// TwinCAT 3 PLC project PLC
// ProgramVersion: 3.1.4023.0
// libraries:
//   Tc2_Standard, * (Beckhoff Automation GmbH)
//   Tc2_System, * (Beckhoff Automation GmbH)
//   Tc3_Module, * (Beckhoff Automation GmbH)
// project tree:
//   / PlcTask.TcTTO
//   POUs/ MAIN.TcPOU
//   DUTs/IO/PdoEntries/ Status_57491DF1.TcDUT, Status_D4FDECD4.TcDUT, Control_0B2F8B70.TcDUT, Status_A3AA621F.TcDUT, Status_B0753356.TcDUT, Status_F2CE6D91.TcDUT, Status_7BCDA921.TcDUT, Ctrl_B9DDD3FF.TcDUT, STATUS_B0753356.TcDUT, Status_8F1D55D8.TcDUT, Status_ACC8459F.TcDUT, Status_3A9E406C.TcDUT, Control_D500AB79.TcDUT, Status_D8D782C3.TcDUT, Control_6EF2C5D0.TcDUT, Status_E2E79E85.TcDUT, Status_E3E7FD12.TcDUT, Status_8CBE219F.TcDUT, Status_B6795845.TcDUT, Control_5FD4673D.TcDUT, Status_1E008DB9.TcDUT, Status_3035BE2E.TcDUT, Control_F189B737.TcDUT, Control_C948E0F2.TcDUT, Status_725F98F2.TcDUT, Device_Diag_1464ECF9.TcDUT, Control_F58A89C5.TcDUT, Status_6CCA259F.TcDUT, Status_72C27E80.TcDUT, Control_254441A5.TcDUT, Status_15ACD201.TcDUT, Device_Status_033C68E9.TcDUT
//   DUTs/IO/PDOs/ InfoData_6F19DB2B.TcDUT, Channel_830843C1.TcDUT, WcState_9091E0EB.TcDUT, ID_Inputs_07C9D28F.TcDUT, InfoData_32EB74EA.TcDUT, Latch_8E413295.TcDUT, WcState_B516A264.TcDUT, InfoData_A7436BC6.TcDUT, CNT_Input_Channel_FF10BD3C.TcDUT, DIG_Inputs_CAFF6004.TcDUT, DIG_Inputs_Device_1F4E72EB.TcDUT, CNT_Output_Channel_550BB6DF.TcDUT, DI_X01_Pin_830843C1.TcDUT, DI_X02_Pin_830843C1.TcDUT, DI_X03_Pin_830843C1.TcDUT, DI_X04_Pin_830843C1.TcDUT, DI_X05_Pin_830843C1.TcDUT, DI_X06_Pin_830843C1.TcDUT, DI_X07_Pin_830843C1.TcDUT, DI_X08_Pin_830843C1.TcDUT, DI_X_830843C1.TcDUT, DIG_Inputs_Channel_ACAA0425.TcDUT, DO_Inputs_Channel_CC455148.TcDUT, DIG_Inputs_Channel_CC455148.TcDUT, DIG_Inputs_Channel_38F9DD27.TcDUT, DIG_Inputs_Device_B3EA4204.TcDUT, AI_Inputs_Channel_C3DE7A0A.TcDUT, DO_X05_Pin_42CA91F7.TcDUT, DO_X06_Pin_42CA91F7.TcDUT, DO_X07_Pin_42CA91F7.TcDUT, DO_X08_Pin_42CA91F7.TcDUT, DO_X_42CA91F7.TcDUT, Group_99EF3D30.TcDUT, Group_8FCDB395.TcDUT, WcState_0B2B16F9.TcDUT, Channel_42CA91F7.TcDUT, Diag_Channel_830843C1.TcDUT, DIG_Inputs_CC455148.TcDUT, DIG_Diag_Inputs_584303BF.TcDUT, DIG_Inputs_Device_E94E5BF9.TcDUT, DIG_Outputs_28AC1A9E.TcDUT, DIG_Outputs_Device_36A5EF17.TcDUT, DO_Inputs_CC455148.TcDUT, DO_Diag_Inputs_584303BF.TcDUT, DO_Inputs_Device_AF161A9E.TcDUT, DO_Outputs_28AC1A9E.TcDUT, DO_Outputs_Device_36A5EF17.TcDUT, DO_Diag_Inputs_CC455148.TcDUT, DO_Diag_Inputs_212B82C1.TcDUT, DIG_Inputs_Device_4E5AF17E.TcDUT, DI_X01_Pin4_Input_830843C1.TcDUT, DI_X01_Pin2_Input_830843C1.TcDUT, DI_X02_Pin4_Input_830843C1.TcDUT, DI_X02_Pin2_Input_830843C1.TcDUT, DO_X03_Pin4_Output_42CA91F7.TcDUT, DO_X03_Pin2_Output_42CA91F7.TcDUT, DO_X04_Pin4_Output_42CA91F7.TcDUT, DO_X04_Pin2_Output_42CA91F7.TcDUT, DI_Inputs_Channel_91AC31B7.TcDUT, DO_Outputs_Channel_28AC1A9E.TcDUT, InfoData_0A66F009.TcDUT, DO_X01_Pin_42CA91F7.TcDUT, DO_X02_Pin_42CA91F7.TcDUT, DO_X03_Pin_42CA91F7.TcDUT, DO_X04_Pin_42CA91F7.TcDUT, DIG_Diag_Inputs_Channel_584303BF.TcDUT, DIG_Output_Channel_28AC1A9E.TcDUT, DO_Inputs_Channel_584303BF.TcDUT, DO_Inputs_Device_4E5AF17E.TcDUT, DIG_Outputs_Channel_28AC1A9E.TcDUT, DIG_Inputs_Device_27CCC866.TcDUT, AI_Standard_Channel_A8DF64E3.TcDUT, DO_Outputs_C0F4C383.TcDUT, AI_Standard_Channel_4A394481.TcDUT, RTD_RTDInputs_Channel_A8DF64E3.TcDUT, TC_TCInputs_Channel_A8DF64E3.TcDUT, AIBridge_Inputs_555AA1E8.TcDUT, AISupply_Inputs_555AA1E8.TcDUT, RMB_Status_C0E100AA.TcDUT, RMB_Value_INT_E9189C4B.TcDUT, RMB_Control_CC49845C.TcDUT, Ch1_Status_75824485.TcDUT, Ch1_Sample_A71DD501.TcDUT, Ch2_Status_75824485.TcDUT, Ch2_Sample_9F6886E6.TcDUT, NextSync1Time_9AFDC275.TcDUT, Sample_Count_EA88CAD9.TcDUT, InfoData_BEF6B88E.TcDUT, DIG_Inputs_697E0EF2.TcDUT, AI_Inputs_Channel_45213104.TcDUT, DEV_Inputs_Device_5F4E175E.TcDUT, DIG_Outputs_DE230DD5.TcDUT, DEV_Outputs_Device_59FFD247.TcDUT, AI_Inputs_Channel_5A86716D.TcDUT, AO_Output_Channel_BA7EBB7C.TcDUT, DI_Inputs_1F3A9325.TcDUT, AI_TxPDO_Map_Standard_Channel_A8DF64E3.TcDUT, AI_Inputs_Channel_A8DF64E3.TcDUT, DI_X03_Pin4_Input_830843C1.TcDUT, DI_X04_Pin4_Input_830843C1.TcDUT, DI_X05_Pin4_Input_830843C1.TcDUT, DI_X06_Pin4_Input_830843C1.TcDUT, DI_X07_Pin4_Input_830843C1.TcDUT, DI_X08_Pin4_Input_830843C1.TcDUT, AI_X01_Pin2_Standard_A8DF64E3.TcDUT, AI_X02_Pin2_Standard_A8DF64E3.TcDUT, AI_X05_Pin2_Standard_A8DF64E3.TcDUT, AI_X06_Pin2_Standard_A8DF64E3.TcDUT, DO_X01_Pin4_Output_42CA91F7.TcDUT, DO_X02_Pin4_Output_42CA91F7.TcDUT, DO_X05_Pin4_Output_42CA91F7.TcDUT, DO_X06_Pin4_Output_42CA91F7.TcDUT, DO_X07_Pin4_Output_42CA91F7.TcDUT, DO_X08_Pin4_Output_42CA91F7.TcDUT, SSI_Inputs_0E3D8E33.TcDUT, ENC_Status_compact_F4F89583.TcDUT, ENC_Control_compact_E6DC9B25.TcDUT, ENC_Status_compact_7D3464F3.TcDUT, ENC_Control_compact_21E2D14D.TcDUT, ENC_Status_compact_4198EF3B.TcDUT, COM_Inputs_6C2FC202.TcDUT, COM_Outputs_5D00B5E7.TcDUT, COM_Inputs_Channel_C252EAC2.TcDUT, COM_Outputs_Channel_B336F4EE.TcDUT, COM_TxPDO_Map_Inputs_Channel_C252EAC2.TcDUT, COM_RxPDO_Map_Outputs_Channel_B336F4EE.TcDUT, COM_TxPDO_Map_Inputs_Channel_6C2FC202.TcDUT, COM_RxPDO_Map_Outputs_Channel_5D00B5E7.TcDUT, DIS_Inputs_E0E384E3.TcDUT, DIS_Outputs_6C9BFFEE.TcDUT, DeviceState_Inputs_Device_A1210598.TcDUT, DeviceState_Inputs_4751FF76.TcDUT, Digital_Inputs_FE042239.TcDUT, InfoData_90184F0C.TcDUT, Module_1_DeviceState_Inputs_Device_5322301C.TcDUT, Module_2_DeviceState_Inputs_BD6C7035.TcDUT, Module_7_Digital_Inputs_F29732B3.TcDUT, Digital_Inputs_8749E151.TcDUT, Module_7_Digital_Inputs_DAAE149B.TcDUT, EMPTY_STRUCTURE.TcDUT, DeviceState_Inputs_C7251DC9.TcDUT, Module_2_DeviceState_Inputs_B92A0D6A.TcDUT, Digital_Inputs_83D7E782.TcDUT, Module_11_Digital_Inputs_33FD8372.TcDUT, Digital_Inputs_3DEC2D27.TcDUT, Module_11_Digital_Inputs_36A01C39.TcDUT, ENC_Status_compact_4D066E1A.TcDUT, STM_Status_36ED096F.TcDUT, STM_Control_BA4CE352.TcDUT, STM_Velocity_A47A3F41.TcDUT, InfoData_8DF4E0C5.TcDUT, InfoData_6538CF5F.TcDUT, STM_Status_DE0D6B37.TcDUT, FB_Position_3FA094ED.TcDUT, DRV_Statusword_9B36FDFC.TcDUT, DRV_Controlword_F3F14721.TcDUT, DRV_Target_velocity_08A9583B.TcDUT, InfoData_96C94FAE.TcDUT, InfoData_6185D47C.TcDUT, DS402_Statusword_9B36FDFC.TcDUT, DS402_Position_actual_value_07DC4C74.TcDUT, DS402_Controlword_F3F14721.TcDUT, DS402_Target_velocity_08A9583B.TcDUT, ENC_Status_compact_Channel_DC559AB0.TcDUT, DCM_Status_Channel_36ED096F.TcDUT, ENC_Control_compact_Channel_2E82BC43.TcDUT, DCM_Control_Channel_5A8B5016.TcDUT, DCM_Velocity_Channel_A47A3F41.TcDUT, InfoData_939F71B6.TcDUT, DI_Inputs_58955D1A.TcDUT, STM_Status_Channel_99D1DFFA.TcDUT, STM_Synchron_info_data_Channel_DD535D91.TcDUT, STM_Inputs_Device_A41D8456.TcDUT, DO_Outputs_A241BD3A.TcDUT, STM_Control_Channel_F193EBCD.TcDUT, STM_Target_Velocity_Channel_E69D8325.TcDUT, TACHO_Single_Shaft_Mode_Input_Channel_C331CA3E.TcDUT, DIG_Inputs_495F5DA4.TcDUT, PWM_Status_77939B11.TcDUT, DEV_Inputs_FBF180A4.TcDUT, TACHO_Output_Channel_600697D9.TcDUT, DIG_Outputs_0E284394.TcDUT, PWM_Control_63F162E4.TcDUT, DPO_Inputs_Channel_BF408C57.TcDUT, DPO_Inputs_Device_9B08D915.TcDUT, DPO_Outputs_Channel_A459B36C.TcDUT, DPO_Outputs_Device_B673A337.TcDUT, DPO_Inputs_Channel_F87663B8.TcDUT, DPO_Inputs_Device_99241EEA.TcDUT, BCT_Inputs_7ACE8FA6.TcDUT, DPO_Inputs_Channel_0E6D6BE5.TcDUT, DPO_Inputs_Device_0C16AFA0.TcDUT, InfoData_E68C61CD.TcDUT, InfoData_2A97D6CF.TcDUT, Inputs_25A0042B.TcDUT, Outputs_2397A10E.TcDUT
//   DUTs/IO/Boxes/ EK1100_1FC0878B.TcDUT, EK1122_1FC0878B.TcDUT, EP1008_78E8D3DD.TcDUT, EP1018_78E8D3DD.TcDUT, EP1098_78E8D3DD.TcDUT, EP1111_837A6B03.TcDUT, EP1122_1FC0878B.TcDUT, EP1258_58F475DD.TcDUT, EP1312_1FC0878B.TcDUT, EP1518_CC442588.TcDUT, EP1809_32157CFD.TcDUT, EP1809_AA84A50E.TcDUT, EP1809_8E14C816.TcDUT, EP1816_73178B54.TcDUT, EP1816_03D88109.TcDUT, EP1816_5E50D3DD.TcDUT, EP1816_F50297FE.TcDUT, EP1816_CABD51E6.TcDUT, EP1819_32157CFD.TcDUT, EP1859_B704EC1A.TcDUT, EP1859_B9D5A785.TcDUT, EP2001_C23D36A6.TcDUT, EP2008_E2806B95.TcDUT, EP2028_E2806B95.TcDUT, EP2038_3AE10DD7.TcDUT, EP2308_F6D9A8D1.TcDUT, EP2316_CAC4656D.TcDUT, EP2316_528F6B1F.TcDUT, EP2316_3C060514.TcDUT, EP2316_DCD24F8F.TcDUT, EP2318_F6D9A8D1.TcDUT, EP2328_F6D9A8D1.TcDUT, EP2328_F66CDDB7.TcDUT, EP2338_39FFBC52.TcDUT, EP2338_7699BCF6.TcDUT, EP2339_B2B612E8.TcDUT, EP2339_C2A6198C.TcDUT, EP2339_D8E9F29A.TcDUT, EP2339_4CF33DED.TcDUT, EP2339_56BCD6FB.TcDUT, EP2339_49541507.TcDUT, EP2339_E3933831.TcDUT, EP2349_4CF33DED.TcDUT, EP2624_7B64371E.TcDUT, EP2809_2B6483BD.TcDUT, EP2809_7AAF2E71.TcDUT, EP2809_23623E9C.TcDUT, EP2816_F9F6AB82.TcDUT, EP2816_88324133.TcDUT, EP2816_0C961E28.TcDUT, EP2816_D9B77CAE.TcDUT, EP2816_01296449.TcDUT, EP2817_7CB3CE29.TcDUT, EP3162_AA20D87B.TcDUT, EP3162_C396CC55.TcDUT, EP3174_C4269E32.TcDUT, EP3174_DCC78662.TcDUT, EP3182_0BD171D7.TcDUT, EP3182_C396CC55.TcDUT, EP3184_C4269E32.TcDUT, EP3184_DCC78662.TcDUT, EP3204_6CD7E119.TcDUT, EP3204_AB25C3AC.TcDUT, EP3314_1CEB931C.TcDUT, EP3314_E65CDB1C.TcDUT, EP3351_6847F283.TcDUT, EP3356_1EAAA6FF.TcDUT, EP3632_E2B98A5C.TcDUT, EP3744_315C92D4.TcDUT, EP3752_C992DA1B.TcDUT, EP4174_AB92710E.TcDUT, EP4314_454AD8BA.TcDUT, EP4374_D4EA2234.TcDUT, EP4374_A304750F.TcDUT, EP4378_34BF187E.TcDUT, EP5001_0B28D087.TcDUT, EP5101_87AC78CF.TcDUT, EP5101_7476E948.TcDUT, EP5151_7476E948.TcDUT, EP5101_382A92AF.TcDUT, EP6001_40883D03.TcDUT, EP6002_2663B0AE.TcDUT, EP6002_7F53816A.TcDUT, EP6002_7BE6B617.TcDUT, EP6090_18BD01E9.TcDUT, EP6224_7D7C361B.TcDUT, EP6224_77EE7830.TcDUT, EP6224_EDFF9F2F.TcDUT, EP6224_98EF2419.TcDUT, EP6228_FB34C737.TcDUT, EP6228_495B58F4.TcDUT, EP6228_C205B548.TcDUT, EP6601_EEB2FEF4.TcDUT, EP7041_9A9CCB1D.TcDUT, EP7041_3210CF40.TcDUT, EP7041_3E4BEAEF.TcDUT, EP7047_3E4BEAEF.TcDUT, EP7211_CE650BCF.TcDUT, EP7211_FC4732E8.TcDUT, EP7211_7BF21317.TcDUT, EP7342_2AE9C6B3.TcDUT, EP7402_190E1004.TcDUT, EP8309_A0C54F77.TcDUT, EP9128_1FC0878B.TcDUT, EP9214_7560C653.TcDUT, EP9224_2E4B686C.TcDUT, EP9521_1FC0878B.TcDUT, EP9576_C42142C6.TcDUT, EP9224_079410B7.TcDUT, EP9224_1FC0878B.TcDUT
//   DUTs/IO/Devices/ SyncUnitTask_2D604ED5.TcDUT, SyncUnitTasks_6FEB8257.TcDUT, SyncUnits_2E61B955.TcDUT
//   DUTs/IO/Topology/ A_0037_EP1312_0001_0016_211442AD.TcDUT (not stored), A_0026_EP1122_0001_0018_73CBC47E.TcDUT (not stored), A_0025_EP1122_0001_0017_496E3A36.TcDUT, A_0024_EP1122_0001_0016_DB5F1CD0.TcDUT, Beckhoff_EP1xxxEK1122_3357DBA9.TcDUT (not stored), Beckhoff_EP1xxx_617026EA.TcDUT (not stored), Beckhoff_EP2xxxEK1122_6A4FE0FF.TcDUT (not stored), Beckhoff_EP2xxx_5E6BC55D.TcDUT (not stored), Beckhoff_EP3xxxEK1122_7B33BCBC.TcDUT (not stored), Beckhoff_EP3xxx_05483C40.TcDUT (not stored), Beckhoff_EP4xxxEK1122_BF2FC8FC.TcDUT (not stored), Beckhoff_EP4xxx_5F57EEFA.TcDUT (not stored), Beckhoff_EP5xxxEK1122_686419BC.TcDUT (not stored), Beckhoff_EP5xxx_7357566B.TcDUT (not stored), Beckhoff_EP6xxxEK1122_67CC26DB.TcDUT (not stored), Beckhoff_EP6xxx_09B4DFD6.TcDUT (not stored), A_0054_EP7402_0057_0017_30592BBB.TcDUT (not stored), Beckhoff_EP7xxxEK1122_5EFC4D75.TcDUT (not stored), Beckhoff_EP7xxx_ED361224.TcDUT (not stored), Beckhoff_EP8xxxEK1122_7348582A.TcDUT (not stored), Beckhoff_EP8xxx_7FC896F3.TcDUT (not stored), A_0024_EP9521_0020_0000_1CEF36B8.TcDUT, A_0022_EP9224_0037_0017_CE247778.TcDUT, A_0013_EP9128_0021_0019_0DE615A6.TcDUT, A_0010_EP9128_0021_0018_C959F4E2.TcDUT, A_0007_EP9128_0021_0017_F9495D48.TcDUT, A_0004_EP9128_0021_0016_EBEEF4C1.TcDUT, A_0001_EP9128_0020_0016_F00690F4.TcDUT, Beckhoff_EP9xxxEK1122_2EAED5FB.TcDUT (not stored), Beckhoff_EP9xxx_0E1CA865.TcDUT (not stored), EtherCAT_Master_EPxxxx_2B438D5B.TcDUT (not stored)
//   DUTs/IO/Base/ EtcSlaveBase_82538BE2.TcDUT, EtcSlaveBase_82538BE2.TcDUT, EtcSlaveBase_82538BE2.TcDUT, EtcSlaveTerminalBase_947E5A46.TcDUT, EtcSlaveBoxBase_77A0E4A7.TcDUT, EtcSlaveEndTerminalBase_866C7F0C.TcDUT, InputBase_8311D824.TcDUT, OutputBase_10CEE7DE.TcDUT, EtcMasterBase_62654B43.TcDUT
//   GVLs/ GVL_iXlinker.TcGVL

CONFIGURATION PLC
    RESOURCE PLC ON TwinCAT3
        TASK PlcTask(INTERVAL := T#10ms, PRIORITY := 20);
        PROGRAM MAIN WITH PlcTask : MAIN;
    END_RESOURCE
END_CONFIGURATION

// ---- DUTs/IO/PdoEntries/Status_57491DF1.TcDUT
{attribute 'GeneratedUsingTerminal: EP1518-0002-0016'}
{attribute addProperty BoxType "EP1518-0002-0016"}
{attribute addProperty Id "Set_counter_doneBOOL1Counter_inhibitedBOOL1Status_of_input_UDBOOL1Status_of_input_clockBOOL1Sync_errorBOOL1TxPDO_StateBOOL1TxPDO_ToggleBOOL1"}
{attribute addProperty CRC "1464409585"}
{attribute addProperty Size "7"}
TYPE Status_57491DF1 :
STRUCT
	{attribute addProperty Name "Set_counter_done"}
	Set_counter_done : BOOL;
	{attribute addProperty Name "Counter_inhibited"}
	Counter_inhibited : BOOL;
	{attribute addProperty Name "Status_of_input_UD"}
	Status_of_input_UD : BOOL;
	{attribute addProperty Name "Status_of_input_clock"}
	Status_of_input_clock : BOOL;
	{attribute addProperty Name "Sync_error"}
	Sync_error : BOOL;
	{attribute addProperty Name "TxPDO_State"}
	TxPDO_State : BOOL;
	{attribute addProperty Name "TxPDO_Toggle"}
	TxPDO_Toggle : BOOL;
END_STRUCT
END_TYPE

// ---- DUTs/IO/PdoEntries/Status_D4FDECD4.TcDUT
{attribute 'GeneratedUsingTerminal: EP1518-0002-0016'}
{attribute addProperty BoxType "EP1518-0002-0016"}
{attribute addProperty Id "Error_channel_1BOOL1Error_channel_2BOOL1Sync_errorBOOL1TxPDO_StateBOOL1TxPDO_ToggleBOOL1"}
{attribute addProperty CRC "3573411028"}
{attribute addProperty Size "5"}
TYPE Status_D4FDECD4 :
STRUCT
	{attribute addProperty Name "Error_channel_1"}
	Error_channel_1 : BOOL;
	{attribute addProperty Name "Error_channel_2"}
	Error_channel_2 : BOOL;
	{attribute addProperty Name "Sync_error"}
	Sync_error : BOOL;
	{attribute addProperty Name "TxPDO_State"}
	TxPDO_State : BOOL;
	{attribute addProperty Name "TxPDO_Toggle"}
	TxPDO_Toggle : BOOL;
END_STRUCT
END_TYPE

// ---- DUTs/IO/PdoEntries/Control_0B2F8B70.TcDUT
{attribute 'GeneratedUsingTerminal: EP1518-0002-0016'}
{attribute addProperty BoxType "EP1518-0002-0016"}
{attribute addProperty Id "Set_counterBOOL1Inhibit_counterBOOL1"}
{attribute addProperty CRC "187665264"}
{attribute addProperty Size "2"}
TYPE Control_0B2F8B70 :
STRUCT
	{attribute addProperty Name "Set_counter"}
	Set_counter : BOOL;
	{attribute addProperty Name "Inhibit_counter"}
	Inhibit_counter : BOOL;
END_STRUCT
END_TYPE

// ---- DUTs/IO/PdoEntries/Status_A3AA621F.TcDUT
{attribute 'GeneratedUsingTerminal: EP1816-3008-0016'}
{attribute addProperty BoxType "EP1816-3008-0016"}
{attribute addProperty Id "ErrorBOOL1TxPDO_ToggleBOOL1"}
{attribute addProperty CRC "2745852447"}
{attribute addProperty Size "2"}
TYPE Status_A3AA621F :
STRUCT
	{attribute addProperty Name "Error"}
	Error : BOOL;
	{attribute addProperty Name "TxPDO_Toggle"}
	TxPDO_Toggle : BOOL;
END_STRUCT
END_TYPE

// ---- DUTs/IO/PdoEntries/Status_B0753356.TcDUT
{attribute 'GeneratedUsingTerminal: EP3632-0001-0016'}
{attribute addProperty BoxType "EP3632-0001-0016"}
{attribute addProperty Id "UnderrangeBOOL1OverrangeBOOL1Limit_1BYTE1Limit_2BYTE1ErrorBOOL1Sync_errorBOOL1TxPDO_StateBOOL1TxPDO_ToggleBOOL1"}
{attribute addProperty CRC "2960470870"}
{attribute addProperty Size "8"}
TYPE STATUS_B0753356 :
STRUCT
	{attribute addProperty Name "Underrange"}
	Underrange : BOOL;
	{attribute addProperty Name "Overrange"}
	Overrange : BOOL;
	{attribute addProperty Name "Limit_1"}
	Limit_1 : BYTE;
	{attribute addProperty Name "Limit_2"}
	Limit_2 : BYTE;
	{attribute addProperty Name "Error"}
	Error : BOOL;
	{attribute addProperty Name "Sync_error"}
	Sync_error : BOOL;
	{attribute addProperty Name "TxPDO_State"}
	TxPDO_State : BOOL;
	{attribute addProperty Name "TxPDO_Toggle"}
	TxPDO_Toggle : BOOL;
END_STRUCT
END_TYPE

// ---- DUTs/IO/PdoEntries/Status_F2CE6D91.TcDUT
{attribute 'GeneratedUsingTerminal: EP3174-0002-0016'}
{attribute addProperty BoxType "EP3174-0002-0016"}
{attribute addProperty Id "UnderrangeBOOL1OverrangeBOOL1Limit_1BYTE1Limit_2BYTE1ErrorBOOL1TxPDO_StateBOOL1TxPDO_ToggleBOOL1"}
{attribute addProperty CRC "4073614737"}
{attribute addProperty Size "7"}
TYPE Status_F2CE6D91 :
STRUCT
	{attribute addProperty Name "Underrange"}
	Underrange : BOOL;
	{attribute addProperty Name "Overrange"}
	Overrange : BOOL;
	{attribute addProperty Name "Limit_1"}
	Limit_1 : BYTE;
	{attribute addProperty Name "Limit_2"}
	Limit_2 : BYTE;
	{attribute addProperty Name "Error"}
	Error : BOOL;
	{attribute addProperty Name "TxPDO_State"}
	TxPDO_State : BOOL;
	{attribute addProperty Name "TxPDO_Toggle"}
	TxPDO_Toggle : BOOL;
END_STRUCT
END_TYPE

// ---- DUTs/IO/PdoEntries/Status_7BCDA921.TcDUT
{attribute 'GeneratedUsingTerminal: EP3356-0022-0016'}
{attribute addProperty BoxType "EP3356-0022-0016"}
{attribute addProperty Id "OverrangeBOOL1Data_invalidBOOL1ErrorBOOL1Calibration_in_progressBOOL1Steady_stateBOOL1Sync_errorBOOL1TxPDO_ToggleBOOL1"}
{attribute addProperty CRC "2077075745"}
{attribute addProperty Size "7"}
TYPE Status_7BCDA921 :
STRUCT
	{attribute addProperty Name "Overrange"}
	Overrange : BOOL;
	{attribute addProperty Name "Data_invalid"}
	Data_invalid : BOOL;
	{attribute addProperty Name "Error"}
	Error : BOOL;
	{attribute addProperty Name "Calibration_in_progress"}
	Calibration_in_progress : BOOL;
	{attribute addProperty Name "Steady_state"}
	Steady_state : BOOL;
	{attribute addProperty Name "Sync_error"}
	Sync_error : BOOL;
	{attribute addProperty Name "TxPDO_Toggle"}
	TxPDO_Toggle : BOOL;
END_STRUCT
END_TYPE

// ---- DUTs/IO/PdoEntries/Ctrl_B9DDD3FF.TcDUT
{attribute 'GeneratedUsingTerminal: EP3356-0022-0016'}
{attribute addProperty BoxType "EP3356-0022-0016"}
{attribute addProperty Id "Start_calibrationBOOL1Disable_calibrationBOOL1Input_freezeBOOL1Sample_modeBOOL1TaraBOOL1"}
{attribute addProperty CRC "3118322687"}
{attribute addProperty Size "5"}
TYPE Ctrl_B9DDD3FF :
STRUCT
	{attribute addProperty Name "Start_calibration"}
	Start_calibration : BOOL;
	{attribute addProperty Name "Disable_calibration"}
	Disable_calibration : BOOL;
	{attribute addProperty Name "Input_freeze"}
	Input_freeze : BOOL;
	{attribute addProperty Name "Sample_mode"}
	Sample_mode : BOOL;
	{attribute addProperty Name "Tara"}
	Tara : BOOL;
END_STRUCT
END_TYPE

// ---- DUTs/IO/PdoEntries/STATUS_B0753356.TcDUT
{attribute 'GeneratedUsingTerminal: EP3632-0001-0016'}
{attribute addProperty BoxType "EP3632-0001-0016"}
{attribute addProperty Id "UnderrangeBOOL1OverrangeBOOL1Limit_1BYTE1Limit_2BYTE1ErrorBOOL1Sync_errorBOOL1TxPDO_StateBOOL1TxPDO_ToggleBOOL1"}
{attribute addProperty CRC "2960470870"}
{attribute addProperty Size "8"}
TYPE STATUS_B0753356 :
STRUCT
	{attribute addProperty Name "Underrange"}
	Underrange : BOOL;
	{attribute addProperty Name "Overrange"}
	Overrange : BOOL;
	{attribute addProperty Name "Limit_1"}
	Limit_1 : BYTE;
	{attribute addProperty Name "Limit_2"}
	Limit_2 : BYTE;
	{attribute addProperty Name "Error"}
	Error : BOOL;
	{attribute addProperty Name "Sync_error"}
	Sync_error : BOOL;
	{attribute addProperty Name "TxPDO_State"}
	TxPDO_State : BOOL;
	{attribute addProperty Name "TxPDO_Toggle"}
	TxPDO_Toggle : BOOL;
END_STRUCT
END_TYPE

// ---- DUTs/IO/PdoEntries/Status_8F1D55D8.TcDUT
{attribute 'GeneratedUsingTerminal: EP3752-0000-0017'}
{attribute addProperty BoxType "EP3752-0000-0017"}
{attribute addProperty Id "ErrorBOOL1TxPDO_StateBOOL1TxPDO_ToggleBOOL1"}
{attribute addProperty CRC "2401064408"}
{attribute addProperty Size "3"}
TYPE Status_8F1D55D8 :
STRUCT
	{attribute addProperty Name "Error"}
	Error : BOOL;
	{attribute addProperty Name "TxPDO_State"}
	TxPDO_State : BOOL;
	{attribute addProperty Name "TxPDO_Toggle"}
	TxPDO_Toggle : BOOL;
END_STRUCT
END_TYPE

// ---- DUTs/IO/PdoEntries/Status_ACC8459F.TcDUT
{attribute 'GeneratedUsingTerminal: EP5001-0002-0016'}
{attribute addProperty BoxType "EP5001-0002-0016"}
{attribute addProperty Id "Data_errorBOOL1Frame_errorBOOL1Power_failureBOOL1Sync_errorBOOL1TxPDO_StateBOOL1TxPDO_ToggleBOOL1"}
{attribute addProperty CRC "2898806175"}
{attribute addProperty Size "6"}
TYPE Status_ACC8459F :
STRUCT
	{attribute addProperty Name "Data_error"}
	Data_error : BOOL;
	{attribute addProperty Name "Frame_error"}
	Frame_error : BOOL;
	{attribute addProperty Name "Power_failure"}
	Power_failure : BOOL;
	{attribute addProperty Name "Sync_error"}
	Sync_error : BOOL;
	{attribute addProperty Name "TxPDO_State"}
	TxPDO_State : BOOL;
	{attribute addProperty Name "TxPDO_Toggle"}
	TxPDO_Toggle : BOOL;
END_STRUCT
END_TYPE

// ---- DUTs/IO/PdoEntries/Status_3A9E406C.TcDUT
{attribute 'GeneratedUsingTerminal: EP5101-0002-0016'}
{attribute addProperty BoxType "EP5101-0002-0016"}
{attribute addProperty Id "Latch_C_validBOOL1Set_counter_doneBOOL1Counter_underflowBOOL1Counter_overflowBOOL1Open_circuitBOOL1Extrapolation_stallBOOL1Status_of_input_ABOOL1Status_of_input_BBOOL1Status_of_input_CBOOL1Sync_errorBOOL1TxPDO_StateBOOL1TxPDO_ToggleBOOL1"}
{attribute addProperty CRC "983449708"}
{attribute addProperty Size "12"}
TYPE Status_3A9E406C :
STRUCT
	{attribute addProperty Name "Latch_C_valid"}
	Latch_C_valid : BOOL;
	{attribute addProperty Name "Set_counter_done"}
	Set_counter_done : BOOL;
	{attribute addProperty Name "Counter_underflow"}
	Counter_underflow : BOOL;
	{attribute addProperty Name "Counter_overflow"}
	Counter_overflow : BOOL;
	{attribute addProperty Name "Open_circuit"}
	Open_circuit : BOOL;
	{attribute addProperty Name "Extrapolation_stall"}
	Extrapolation_stall : BOOL;
	{attribute addProperty Name "Status_of_input_A"}
	Status_of_input_A : BOOL;
	{attribute addProperty Name "Status_of_input_B"}
	Status_of_input_B : BOOL;
	{attribute addProperty Name "Status_of_input_C"}
	Status_of_input_C : BOOL;
	{attribute addProperty Name "Sync_error"}
	Sync_error : BOOL;
	{attribute addProperty Name "TxPDO_State"}
	TxPDO_State : BOOL;
	{attribute addProperty Name "TxPDO_Toggle"}
	TxPDO_Toggle : BOOL;
END_STRUCT
END_TYPE

// ---- DUTs/IO/PdoEntries/Control_D500AB79.TcDUT
{attribute 'GeneratedUsingTerminal: EP5101-0002-0016'}
{attribute addProperty BoxType "EP5101-0002-0016"}
{attribute addProperty Id "Enable_latch_CBOOL1Set_counterBOOL1"}
{attribute addProperty CRC "3573590905"}
{attribute addProperty Size "2"}
TYPE Control_D500AB79 :
STRUCT
	{attribute addProperty Name "Enable_latch_C"}
	Enable_latch_C : BOOL;
	{attribute addProperty Name "Set_counter"}
	Set_counter : BOOL;
END_STRUCT
END_TYPE

// ---- DUTs/IO/PdoEntries/Status_D8D782C3.TcDUT
{attribute 'GeneratedUsingTerminal: EP5101-0011-0016'}
{attribute addProperty BoxType "EP5101-0011-0016"}
{attribute addProperty Id "Latch_C_validBOOL1Latch_extern_validBOOL1Set_counter_doneBOOL1Counter_underflowBOOL1Counter_overflowBOOL1Status_of_input_statusBOOL1Open_circuitBOOL1Extrapolation_stallBOOL1Status_of_input_ABOOL1Status_of_input_BBOOL1Status_of_input_CBOOL1Status_of_input_gateBOOL1Status_of_extern_latchBOOL1Sync_errorBOOL1TxPDO_StateBOOL1TxPDO_ToggleBOOL1"}
{attribute addProperty CRC "3638002371"}
{attribute addProperty Size "16"}
TYPE Status_D8D782C3 :
STRUCT
	{attribute addProperty Name "Latch_C_valid"}
	Latch_C_valid : BOOL;
	{attribute addProperty Name "Latch_extern_valid"}
	Latch_extern_valid : BOOL;
	{attribute addProperty Name "Set_counter_done"}
	Set_counter_done : BOOL;
	{attribute addProperty Name "Counter_underflow"}
	Counter_underflow : BOOL;
	{attribute addProperty Name "Counter_overflow"}
	Counter_overflow : BOOL;
	{attribute addProperty Name "Status_of_input_status"}
	Status_of_input_status : BOOL;
	{attribute addProperty Name "Open_circuit"}
	Open_circuit : BOOL;
	{attribute addProperty Name "Extrapolation_stall"}
	Extrapolation_stall : BOOL;
	{attribute addProperty Name "Status_of_input_A"}
	Status_of_input_A : BOOL;
	{attribute addProperty Name "Status_of_input_B"}
	Status_of_input_B : BOOL;
	{attribute addProperty Name "Status_of_input_C"}
	Status_of_input_C : BOOL;
	{attribute addProperty Name "Status_of_input_gate"}
	Status_of_input_gate : BOOL;
	{attribute addProperty Name "Status_of_extern_latch"}
	Status_of_extern_latch : BOOL;
	{attribute addProperty Name "Sync_error"}
	Sync_error : BOOL;
	{attribute addProperty Name "TxPDO_State"}
	TxPDO_State : BOOL;
	{attribute addProperty Name "TxPDO_Toggle"}
	TxPDO_Toggle : BOOL;
END_STRUCT
END_TYPE

// ---- DUTs/IO/PdoEntries/Control_6EF2C5D0.TcDUT
{attribute 'GeneratedUsingTerminal: EP5101-0011-0016'}
{attribute addProperty BoxType "EP5101-0011-0016"}
{attribute addProperty Id "Enable_latch_CBOOL1Enable_latch_extern_on_positive_edgeBOOL1Set_counterBOOL1Enable_latch_extern_on_negative_edgeBOOL1"}
{attribute addProperty CRC "1861404112"}
{attribute addProperty Size "4"}
TYPE Control_6EF2C5D0 :
STRUCT
	{attribute addProperty Name "Enable_latch_C"}
	Enable_latch_C : BOOL;
	{attribute addProperty Name "Enable_latch_extern_on_positive_edge"}
	Enable_latch_extern_on_positive_edge : BOOL;
	{attribute addProperty Name "Set_counter"}
	Set_counter : BOOL;
	{attribute addProperty Name "Enable_latch_extern_on_negative_edge"}
	Enable_latch_extern_on_negative_edge : BOOL;
END_STRUCT
END_TYPE

// ---- DUTs/IO/PdoEntries/Status_E2E79E85.TcDUT
{attribute 'GeneratedUsingTerminal: EP5101-2011-0016'}
{attribute addProperty BoxType "EP5101-2011-0016"}
{attribute addProperty Id "Latch_C_validBOOL1Latch_extern_validBOOL1Set_counter_doneBOOL1Status_of_input_statusBOOL1Open_circuitBOOL1Status_of_input_ABOOL1Status_of_input_BBOOL1Status_of_input_CBOOL1Status_of_input_gateBOOL1Status_of_extern_latchBOOL1Sync_errorBOOL1TxPDO_StateBOOL1TxPDO_ToggleBOOL1"}
{attribute addProperty CRC "3806830213"}
{attribute addProperty Size "13"}
TYPE Status_E2E79E85 :
STRUCT
	{attribute addProperty Name "Latch_C_valid"}
	Latch_C_valid : BOOL;
	{attribute addProperty Name "Latch_extern_valid"}
	Latch_extern_valid : BOOL;
	{attribute addProperty Name "Set_counter_done"}
	Set_counter_done : BOOL;
	{attribute addProperty Name "Status_of_input_status"}
	Status_of_input_status : BOOL;
	{attribute addProperty Name "Open_circuit"}
	Open_circuit : BOOL;
	{attribute addProperty Name "Status_of_input_A"}
	Status_of_input_A : BOOL;
	{attribute addProperty Name "Status_of_input_B"}
	Status_of_input_B : BOOL;
	{attribute addProperty Name "Status_of_input_C"}
	Status_of_input_C : BOOL;
	{attribute addProperty Name "Status_of_input_gate"}
	Status_of_input_gate : BOOL;
	{attribute addProperty Name "Status_of_extern_latch"}
	Status_of_extern_latch : BOOL;
	{attribute addProperty Name "Sync_error"}
	Sync_error : BOOL;
	{attribute addProperty Name "TxPDO_State"}
	TxPDO_State : BOOL;
	{attribute addProperty Name "TxPDO_Toggle"}
	TxPDO_Toggle : BOOL;
END_STRUCT
END_TYPE

// ---- DUTs/IO/PdoEntries/Status_E3E7FD12.TcDUT
{attribute 'GeneratedUsingTerminal: EP6090-0000-0017'}
{attribute addProperty BoxType "EP6090-0000-0017"}
{attribute addProperty Id "UpBOOL1DownBOOL1LeftBOOL1RightBOOL1EnterBOOL1TxPDO_ToggleBOOL1"}
{attribute addProperty CRC "3823631634"}
{attribute addProperty Size "6"}
TYPE Status_E3E7FD12 :
STRUCT
	{attribute addProperty Name "Up"}
	Up : BOOL;
	{attribute addProperty Name "Down"}
	Down : BOOL;
	{attribute addProperty Name "Left"}
	Left : BOOL;
	{attribute addProperty Name "Right"}
	Right : BOOL;
	{attribute addProperty Name "Enter"}
	Enter : BOOL;
	{attribute addProperty Name "TxPDO_Toggle"}
	TxPDO_Toggle : BOOL;
END_STRUCT
END_TYPE

// ---- DUTs/IO/PdoEntries/Status_8CBE219F.TcDUT
{attribute 'GeneratedUsingTerminal: EP7041-0002-0016'}
{attribute addProperty BoxType "EP7041-0002-0016"}
{attribute addProperty Id "Latch_C_validBOOL1Latch_extern_validBOOL1Set_counter_doneBOOL1Counter_underflowBOOL1Counter_overflowBOOL1Extrapolation_stallBOOL1Status_of_input_ABOOL1Status_of_input_BBOOL1Status_of_input_CBOOL1Status_of_extern_latchBOOL1Sync_errorBOOL1TxPDO_ToggleBOOL1"}
{attribute addProperty CRC "2361270687"}
{attribute addProperty Size "12"}
TYPE Status_8CBE219F :
STRUCT
	{attribute addProperty Name "Latch_C_valid"}
	Latch_C_valid : BOOL;
	{attribute addProperty Name "Latch_extern_valid"}
	Latch_extern_valid : BOOL;
	{attribute addProperty Name "Set_counter_done"}
	Set_counter_done : BOOL;
	{attribute addProperty Name "Counter_underflow"}
	Counter_underflow : BOOL;
	{attribute addProperty Name "Counter_overflow"}
	Counter_overflow : BOOL;
	{attribute addProperty Name "Extrapolation_stall"}
	Extrapolation_stall : BOOL;
	{attribute addProperty Name "Status_of_input_A"}
	Status_of_input_A : BOOL;
	{attribute addProperty Name "Status_of_input_B"}
	Status_of_input_B : BOOL;
	{attribute addProperty Name "Status_of_input_C"}
	Status_of_input_C : BOOL;
	{attribute addProperty Name "Status_of_extern_latch"}
	Status_of_extern_latch : BOOL;
	{attribute addProperty Name "Sync_error"}
	Sync_error : BOOL;
	{attribute addProperty Name "TxPDO_Toggle"}
	TxPDO_Toggle : BOOL;
END_STRUCT
END_TYPE

// ---- DUTs/IO/PdoEntries/Status_B6795845.TcDUT
{attribute 'GeneratedUsingTerminal: EP7041-0002-0016'}
{attribute addProperty BoxType "EP7041-0002-0016"}
{attribute addProperty Id "Ready_to_enableBOOL1ReadyBOOL1WarningBOOL1ErrorBOOL1Moving_positiveBOOL1Moving_negativeBOOL1Torque_reducedBOOL1Digital_input_1BOOL1Digital_input_2BOOL1Sync_errorBOOL1TxPDO_ToggleBOOL1"}
{attribute addProperty CRC "3061405765"}
{attribute addProperty Size "11"}
TYPE Status_B6795845 :
STRUCT
	{attribute addProperty Name "Ready_to_enable"}
	Ready_to_enable : BOOL;
	{attribute addProperty Name "Ready"}
	Ready : BOOL;
	{attribute addProperty Name "Warning"}
	Warning : BOOL;
	{attribute addProperty Name "Error"}
	Error : BOOL;
	{attribute addProperty Name "Moving_positive"}
	Moving_positive : BOOL;
	{attribute addProperty Name "Moving_negative"}
	Moving_negative : BOOL;
	{attribute addProperty Name "Torque_reduced"}
	Torque_reduced : BOOL;
	{attribute addProperty Name "Digital_input_1"}
	Digital_input_1 : BOOL;
	{attribute addProperty Name "Digital_input_2"}
	Digital_input_2 : BOOL;
	{attribute addProperty Name "Sync_error"}
	Sync_error : BOOL;
	{attribute addProperty Name "TxPDO_Toggle"}
	TxPDO_Toggle : BOOL;
END_STRUCT
END_TYPE

// ---- DUTs/IO/PdoEntries/Control_5FD4673D.TcDUT
{attribute 'GeneratedUsingTerminal: EP7041-0002-0016'}
{attribute addProperty BoxType "EP7041-0002-0016"}
{attribute addProperty Id "EnableBOOL1ResetBOOL1Reduce_torqueBOOL1Digital_output_1BOOL1"}
{attribute addProperty CRC "1607755581"}
{attribute addProperty Size "4"}
TYPE Control_5FD4673D :
STRUCT
	{attribute addProperty Name "Enable"}
	Enable : BOOL;
	{attribute addProperty Name "Reset"}
	Reset : BOOL;
	{attribute addProperty Name "Reduce_torque"}
	Reduce_torque : BOOL;
	{attribute addProperty Name "Digital_output_1"}
	Digital_output_1 : BOOL;
END_STRUCT
END_TYPE

// ---- DUTs/IO/PdoEntries/Status_1E008DB9.TcDUT
{attribute 'GeneratedUsingTerminal: EP7041-3002-0016'}
{attribute addProperty BoxType "EP7041-3002-0016"}
{attribute addProperty Id "Ready_to_enableBOOL1ReadyBOOL1WarningBOOL1ErrorBOOL1Moving_positiveBOOL1Moving_negativeBOOL1Torque_reducedBOOL1Motor_stallBOOL1Digital_input_1BOOL1Digital_input_2BOOL1Sync_errorBOOL1TxPDO_ToggleBOOL1"}
{attribute addProperty CRC "503352761"}
{attribute addProperty Size "12"}
TYPE Status_1E008DB9 :
STRUCT
	{attribute addProperty Name "Ready_to_enable"}
	Ready_to_enable : BOOL;
	{attribute addProperty Name "Ready"}
	Ready : BOOL;
	{attribute addProperty Name "Warning"}
	Warning : BOOL;
	{attribute addProperty Name "Error"}
	Error : BOOL;
	{attribute addProperty Name "Moving_positive"}
	Moving_positive : BOOL;
	{attribute addProperty Name "Moving_negative"}
	Moving_negative : BOOL;
	{attribute addProperty Name "Torque_reduced"}
	Torque_reduced : BOOL;
	{attribute addProperty Name "Motor_stall"}
	Motor_stall : BOOL;
	{attribute addProperty Name "Digital_input_1"}
	Digital_input_1 : BOOL;
	{attribute addProperty Name "Digital_input_2"}
	Digital_input_2 : BOOL;
	{attribute addProperty Name "Sync_error"}
	Sync_error : BOOL;
	{attribute addProperty Name "TxPDO_Toggle"}
	TxPDO_Toggle : BOOL;
END_STRUCT
END_TYPE

// ---- DUTs/IO/PdoEntries/Status_3035BE2E.TcDUT
{attribute 'GeneratedUsingTerminal: EP7342-0002-0016'}
{attribute addProperty BoxType "EP7342-0002-0016"}
{attribute addProperty Id "Latch_extern_validBOOL1Set_counter_doneBOOL1Counter_underflowBOOL1Counter_overflowBOOL1Extrapolation_stallBOOL1Status_of_input_ABOOL1Status_of_input_BBOOL1Status_of_extern_latchBOOL1Sync_errorBOOL1TxPDO_ToggleBOOL1"}
{attribute addProperty CRC "808828462"}
{attribute addProperty Size "10"}
TYPE Status_3035BE2E :
STRUCT
	{attribute addProperty Name "Latch_extern_valid"}
	Latch_extern_valid : BOOL;
	{attribute addProperty Name "Set_counter_done"}
	Set_counter_done : BOOL;
	{attribute addProperty Name "Counter_underflow"}
	Counter_underflow : BOOL;
	{attribute addProperty Name "Counter_overflow"}
	Counter_overflow : BOOL;
	{attribute addProperty Name "Extrapolation_stall"}
	Extrapolation_stall : BOOL;
	{attribute addProperty Name "Status_of_input_A"}
	Status_of_input_A : BOOL;
	{attribute addProperty Name "Status_of_input_B"}
	Status_of_input_B : BOOL;
	{attribute addProperty Name "Status_of_extern_latch"}
	Status_of_extern_latch : BOOL;
	{attribute addProperty Name "Sync_error"}
	Sync_error : BOOL;
	{attribute addProperty Name "TxPDO_Toggle"}
	TxPDO_Toggle : BOOL;
END_STRUCT
END_TYPE

// ---- DUTs/IO/PdoEntries/Control_F189B737.TcDUT
{attribute 'GeneratedUsingTerminal: EP7342-0002-0016'}
{attribute addProperty BoxType "EP7342-0002-0016"}
{attribute addProperty Id "Enable_latch_extern_on_positive_edgeBOOL1Set_counterBOOL1Enable_latch_extern_on_negative_edgeBOOL1"}
{attribute addProperty CRC "4052334391"}
{attribute addProperty Size "3"}
TYPE Control_F189B737 :
STRUCT
	{attribute addProperty Name "Enable_latch_extern_on_positive_edge"}
	Enable_latch_extern_on_positive_edge : BOOL;
	{attribute addProperty Name "Set_counter"}
	Set_counter : BOOL;
	{attribute addProperty Name "Enable_latch_extern_on_negative_edge"}
	Enable_latch_extern_on_negative_edge : BOOL;
END_STRUCT
END_TYPE

// ---- DUTs/IO/PdoEntries/Control_C948E0F2.TcDUT
{attribute 'GeneratedUsingTerminal: EP7342-0002-0016'}
{attribute addProperty BoxType "EP7342-0002-0016"}
{attribute addProperty Id "EnableBOOL1ResetBOOL1Reduce_torqueBOOL1"}
{attribute addProperty CRC "3376996594"}
{attribute addProperty Size "3"}
TYPE Control_C948E0F2 :
STRUCT
	{attribute addProperty Name "Enable"}
	Enable : BOOL;
	{attribute addProperty Name "Reset"}
	Reset : BOOL;
	{attribute addProperty Name "Reduce_torque"}
	Reduce_torque : BOOL;
END_STRUCT
END_TYPE

// ---- DUTs/IO/PdoEntries/Status_725F98F2.TcDUT
{attribute 'GeneratedUsingTerminal: EP7402-0057-0017'}
{attribute addProperty BoxType "EP7402-0057-0017"}
{attribute addProperty Id "Ready_to_enableBOOL1ReadyBOOL1WarningBOOL1ErrorBOOL1Moving_positiveBOOL1Moving_negativeBOOL1TxPDO_ToggleBOOL1"}
{attribute addProperty CRC "1918867698"}
{attribute addProperty Size "7"}
TYPE Status_725F98F2 :
STRUCT
	{attribute addProperty Name "Ready_to_enable"}
	Ready_to_enable : BOOL;
	{attribute addProperty Name "Ready"}
	Ready : BOOL;
	{attribute addProperty Name "Warning"}
	Warning : BOOL;
	{attribute addProperty Name "Error"}
	Error : BOOL;
	{attribute addProperty Name "Moving_positive"}
	Moving_positive : BOOL;
	{attribute addProperty Name "Moving_negative"}
	Moving_negative : BOOL;
	{attribute addProperty Name "TxPDO_Toggle"}
	TxPDO_Toggle : BOOL;
END_STRUCT
END_TYPE

// ---- DUTs/IO/PdoEntries/Device_Diag_1464ECF9.TcDUT
{attribute 'GeneratedUsingTerminal: EP7402-0057-0017'}
{attribute addProperty BoxType "EP7402-0057-0017"}
{attribute addProperty Id "Device_undervoltageBOOL1Device_overvoltageBOOL1Overtemperature_warningBOOL1Overtemperature_errorBOOL1General_hardware_errorBOOL1Channel_1_openloadBOOL1Channel_1_short_circuitBOOL1Channel_1_motor_overload_I2T_warningBOOL1Channel_1_motor_overload_I2T_errorBOOL1Channel_1_amplifier_overload_I2T_warningBOOL1Channel_1_amplifier_overload_I2T_errorBOOL1Channel_1_in_limit_xBOOL1Channel_1_commutation_errorBOOL1Channel_2_openloadBOOL1Channel_2_short_circuitBOOL1Channel_2_motor_overload_I2T_warningBOOL1Channel_2_motor_overload_I2T_errorBOOL1Channel_2_amplifier_overload_I2T_warningBOOL1Channel_2_amplifier_overload_I2T_errorBOOL1Channel_2_in_limit_xBOOL1Channel_2_commutation_errorBOOL1"}
{attribute addProperty CRC "342158585"}
{attribute addProperty Size "21"}
TYPE Device_Diag_1464ECF9 :
STRUCT
	{attribute addProperty Name "Device_undervoltage"}
	Device_undervoltage : BOOL;
	{attribute addProperty Name "Device_overvoltage"}
	Device_overvoltage : BOOL;
	{attribute addProperty Name "Overtemperature_warning"}
	Overtemperature_warning : BOOL;
	{attribute addProperty Name "Overtemperature_error"}
	Overtemperature_error : BOOL;
	{attribute addProperty Name "General_hardware_error"}
	General_hardware_error : BOOL;
	{attribute addProperty Name "Channel_1_openload"}
	Channel_1_openload : BOOL;
	{attribute addProperty Name "Channel_1_short_circuit"}
	Channel_1_short_circuit : BOOL;
	{attribute addProperty Name "Channel_1_motor_overload_I2T_warning"}
	Channel_1_motor_overload_I2T_warning : BOOL;
	{attribute addProperty Name "Channel_1_motor_overload_I2T_error"}
	Channel_1_motor_overload_I2T_error : BOOL;
	{attribute addProperty Name "Channel_1_amplifier_overload_I2T_warning"}
	Channel_1_amplifier_overload_I2T_warning : BOOL;
	{attribute addProperty Name "Channel_1_amplifier_overload_I2T_error"}
	Channel_1_amplifier_overload_I2T_error : BOOL;
	{attribute addProperty Name "Channel_1_in_limit_x"}
	Channel_1_in_limit_x : BOOL;
	{attribute addProperty Name "Channel_1_commutation_error"}
	Channel_1_commutation_error : BOOL;
	{attribute addProperty Name "Channel_2_openload"}
	Channel_2_openload : BOOL;
	{attribute addProperty Name "Channel_2_short_circuit"}
	Channel_2_short_circuit : BOOL;
	{attribute addProperty Name "Channel_2_motor_overload_I2T_warning"}
	Channel_2_motor_overload_I2T_warning : BOOL;
	{attribute addProperty Name "Channel_2_motor_overload_I2T_error"}
	Channel_2_motor_overload_I2T_error : BOOL;
	{attribute addProperty Name "Channel_2_amplifier_overload_I2T_warning"}
	Channel_2_amplifier_overload_I2T_warning : BOOL;
	{attribute addProperty Name "Channel_2_amplifier_overload_I2T_error"}
	Channel_2_amplifier_overload_I2T_error : BOOL;
	{attribute addProperty Name "Channel_2_in_limit_x"}
	Channel_2_in_limit_x : BOOL;
	{attribute addProperty Name "Channel_2_commutation_error"}
	Channel_2_commutation_error : BOOL;
END_STRUCT
END_TYPE

// ---- DUTs/IO/PdoEntries/Control_F58A89C5.TcDUT
{attribute 'GeneratedUsingTerminal: EP7402-0057-0017'}
{attribute addProperty BoxType "EP7402-0057-0017"}
{attribute addProperty Id "EnableBOOL1ResetBOOL1Invert_directionBOOL1Brake_outputBOOL1"}
{attribute addProperty CRC "4119497157"}
{attribute addProperty Size "4"}
TYPE Control_F58A89C5 :
STRUCT
	{attribute addProperty Name "Enable"}
	Enable : BOOL;
	{attribute addProperty Name "Reset"}
	Reset : BOOL;
	{attribute addProperty Name "Invert_direction"}
	Invert_direction : BOOL;
	{attribute addProperty Name "Brake_output"}
	Brake_output : BOOL;
END_STRUCT
END_TYPE

// ---- DUTs/IO/PdoEntries/Status_6CCA259F.TcDUT
{attribute 'GeneratedUsingTerminal: EP8309-0022-0021'}
{attribute addProperty BoxType "EP8309-0022-0021"}
{attribute addProperty Id "Error_Input_ABOOL1Input_Status_ABOOL1Error_Input_BBOOL1Input_Status_BBOOL1Speed_Below_ThresholdBOOL1TxPDO_ToggleBOOL1"}
{attribute addProperty CRC "1825187231"}
{attribute addProperty Size "6"}
TYPE Status_6CCA259F :
STRUCT
	{attribute addProperty Name "Error_Input_A"}
	Error_Input_A : BOOL;
	{attribute addProperty Name "Input_Status_A"}
	Input_Status_A : BOOL;
	{attribute addProperty Name "Error_Input_B"}
	Error_Input_B : BOOL;
	{attribute addProperty Name "Input_Status_B"}
	Input_Status_B : BOOL;
	{attribute addProperty Name "Speed_Below_Threshold"}
	Speed_Below_Threshold : BOOL;
	{attribute addProperty Name "TxPDO_Toggle"}
	TxPDO_Toggle : BOOL;
END_STRUCT
END_TYPE

// ---- DUTs/IO/PdoEntries/Status_72C27E80.TcDUT
{attribute 'GeneratedUsingTerminal: EP8309-0022-0021'}
{attribute addProperty BoxType "EP8309-0022-0021"}
{attribute addProperty Id "Ready_to_enableBOOL1WarningBOOL1ErrorBOOL1TxPDO_ToggleBOOL1"}
{attribute addProperty CRC "1925348992"}
{attribute addProperty Size "4"}
TYPE Status_72C27E80 :
STRUCT
	{attribute addProperty Name "Ready_to_enable"}
	Ready_to_enable : BOOL;
	{attribute addProperty Name "Warning"}
	Warning : BOOL;
	{attribute addProperty Name "Error"}
	Error : BOOL;
	{attribute addProperty Name "TxPDO_Toggle"}
	TxPDO_Toggle : BOOL;
END_STRUCT
END_TYPE

// ---- DUTs/IO/PdoEntries/Control_254441A5.TcDUT
{attribute 'GeneratedUsingTerminal: EP8309-0022-0021'}
{attribute addProperty BoxType "EP8309-0022-0021"}
{attribute addProperty Id "Enable_ditheringBOOL1EnableBOOL1ResetBOOL1"}
{attribute addProperty CRC "625230245"}
{attribute addProperty Size "3"}
TYPE Control_254441A5 :
STRUCT
	{attribute addProperty Name "Enable_dithering"}
	Enable_dithering : BOOL;
	{attribute addProperty Name "Enable"}
	Enable : BOOL;
	{attribute addProperty Name "Reset"}
	Reset : BOOL;
END_STRUCT
END_TYPE

// ---- DUTs/IO/PdoEntries/Status_15ACD201.TcDUT
{attribute 'GeneratedUsingTerminal: EP9224-0037-0017'}
{attribute addProperty BoxType "EP9224-0037-0017"}
{attribute addProperty Id "Error_UsBOOL1Error_UpBOOL1Warning_UsBOOL1Warning_UpBOOL1Status_UsBOOL1Status_UpBOOL1Channel_ErrorBOOL1Error_Sum_CurrentBOOL1Warning_Sum_CurrentBOOL1TxPDO_StateBOOL1TxPDO_ToggleBOOL1"}
{attribute addProperty CRC "363647489"}
{attribute addProperty Size "11"}
TYPE Status_15ACD201 :
STRUCT
	{attribute addProperty Name "Error_Us"}
	Error_Us : BOOL;
	{attribute addProperty Name "Error_Up"}
	Error_Up : BOOL;
	{attribute addProperty Name "Warning_Us"}
	Warning_Us : BOOL;
	{attribute addProperty Name "Warning_Up"}
	Warning_Up : BOOL;
	{attribute addProperty Name "Status_Us"}
	Status_Us : BOOL;
	{attribute addProperty Name "Status_Up"}
	Status_Up : BOOL;
	{attribute addProperty Name "Channel_Error"}
	Channel_Error : BOOL;
	{attribute addProperty Name "Error_Sum_Current"}
	Error_Sum_Current : BOOL;
	{attribute addProperty Name "Warning_Sum_Current"}
	Warning_Sum_Current : BOOL;
	{attribute addProperty Name "TxPDO_State"}
	TxPDO_State : BOOL;
	{attribute addProperty Name "TxPDO_Toggle"}
	TxPDO_Toggle : BOOL;
END_STRUCT
END_TYPE

// ---- DUTs/IO/PdoEntries/Device_Status_033C68E9.TcDUT
{attribute 'GeneratedUsingTerminal: EP9224-0037-0017'}
{attribute addProperty BoxType "EP9224-0037-0017"}
{attribute addProperty Id "Warning_TemperatureBOOL1Error_TemperatureBOOL1Warning_UsBOOL1Error_UsBOOL1Warning_UpBOOL1Error_UpBOOL1Global_Error_BitBOOL1Warning_Sum_CurrentBOOL1Error_Sum_CurrentBOOL1TxPDO_StateBOOL1TxPDO_ToggleBOOL1"}
{attribute addProperty CRC "54290665"}
{attribute addProperty Size "11"}
TYPE Device_Status_033C68E9 :
STRUCT
	{attribute addProperty Name "Warning_Temperature"}
	Warning_Temperature : BOOL;
	{attribute addProperty Name "Error_Temperature"}
	Error_Temperature : BOOL;
	{attribute addProperty Name "Warning_Us"}
	Warning_Us : BOOL;
	{attribute addProperty Name "Error_Us"}
	Error_Us : BOOL;
	{attribute addProperty Name "Warning_Up"}
	Warning_Up : BOOL;
	{attribute addProperty Name "Error_Up"}
	Error_Up : BOOL;
	{attribute addProperty Name "Global_Error_Bit"}
	Global_Error_Bit : BOOL;
	{attribute addProperty Name "Warning_Sum_Current"}
	Warning_Sum_Current : BOOL;
	{attribute addProperty Name "Error_Sum_Current"}
	Error_Sum_Current : BOOL;
	{attribute addProperty Name "TxPDO_State"}
	TxPDO_State : BOOL;
	{attribute addProperty Name "TxPDO_Toggle"}
	TxPDO_Toggle : BOOL;
END_STRUCT
END_TYPE

// ---- DUTs/IO/PDOs/InfoData_6F19DB2B.TcDUT
{attribute 'GeneratedUsingTerminal: EK1100-0000-0018'}
{attribute addProperty BoxType "EK1100-0000-0018"}
{attribute addProperty Id "StateAT %I*UINT2"}
{attribute addProperty CRC "1863965483"}
{attribute addProperty Size "2"}
TYPE InfoData_6F19DB2B :
STRUCT
	{attribute addProperty Name "State"}
	State AT %I* : UINT;
END_STRUCT
END_TYPE

// ---- DUTs/IO/PDOs/Channel_830843C1.TcDUT
{attribute 'GeneratedUsingTerminal: EP1008-0001-0016'}
{attribute addProperty BoxType "EP1008-0001-0016"}
{attribute addProperty Id "InputAT %I*BOOL1"}
{attribute addProperty CRC "2198356929"}
{attribute addProperty Size "1"}
TYPE Channel_830843C1 EXTENDS InputBase_8311D824 :
STRUCT
	{attribute addProperty Name "Input"}
	Input AT %I* : BOOL;
END_STRUCT
END_TYPE

// ---- DUTs/IO/PDOs/WcState_9091E0EB.TcDUT
{attribute 'GeneratedUsingTerminal: EP1008-0001-0016'}
{attribute addProperty BoxType "EP1008-0001-0016"}
{attribute addProperty Id "WcStateAT %I*BOOL1InputToggleAT %I*BOOL1"}
{attribute addProperty CRC "2425479403"}
{attribute addProperty Size "2"}
TYPE WcState_9091E0EB :
STRUCT
	{attribute addProperty Name "WcState"}
	WcState AT %I* : BOOL;
	{attribute addProperty Name "InputToggle"}
	InputToggle AT %I* : BOOL;
END_STRUCT
END_TYPE

// ---- DUTs/IO/PDOs/ID_Inputs_07C9D28F.TcDUT
{attribute 'GeneratedUsingTerminal: EP1111-0000-0016'}
{attribute addProperty BoxType "EP1111-0000-0016"}
{attribute addProperty Id "IDAT %I*UINT2"}
{attribute addProperty CRC "130667151"}
{attribute addProperty Size "2"}
TYPE ID_Inputs_07C9D28F EXTENDS InputBase_8311D824 :
STRUCT
	{attribute addProperty Name "ID"}
	ID AT %I* : UINT;
END_STRUCT
END_TYPE

// ---- DUTs/IO/PDOs/InfoData_32EB74EA.TcDUT
{attribute 'GeneratedUsingTerminal: EP1111-0000-0016'}
{attribute addProperty BoxType "EP1111-0000-0016"}
{attribute addProperty Id "AdsAddrAT %I*AMSADDR8StateAT %I*UINT2"}
{attribute addProperty CRC "854291690"}
{attribute addProperty Size "10"}
TYPE InfoData_32EB74EA EXTENDS InputBase_8311D824 :
STRUCT
	{attribute addProperty Name "AdsAddr"}
	AdsAddr AT %I* : AMSADDR;
	{attribute addProperty Name "State"}
	State AT %I* : UINT;
END_STRUCT
END_TYPE

// ---- DUTs/IO/PDOs/Latch_8E413295.TcDUT
{attribute 'GeneratedUsingTerminal: EP1258-0001-0016'}
{attribute addProperty BoxType "EP1258-0001-0016"}
{attribute addProperty Id "Status0AT %I*USINT1Status1AT %I*USINT1LatchPos0AT %I*ULINT8LatchNeg0AT %I*ULINT8LatchPos1AT %I*ULINT8LatchNeg1AT %I*ULINT8"}
{attribute addProperty CRC "2386637461"}
{attribute addProperty Size "34"}
TYPE Latch_8E413295 EXTENDS InputBase_8311D824 :
STRUCT
	{attribute addProperty Name "Status0"}
	Status0 AT %I* : USINT;
	{attribute addProperty Name "Status1"}
	Status1 AT %I* : USINT;
	{attribute addProperty Name "LatchPos0"}
	LatchPos0 AT %I* : ULINT;
	{attribute addProperty Name "LatchNeg0"}
	LatchNeg0 AT %I* : ULINT;
	{attribute addProperty Name "LatchPos1"}
	LatchPos1 AT %I* : ULINT;
	{attribute addProperty Name "LatchNeg1"}
	LatchNeg1 AT %I* : ULINT;
END_STRUCT
END_TYPE

// ---- DUTs/IO/PDOs/WcState_B516A264.TcDUT
{attribute 'GeneratedUsingTerminal: EP1258-0001-0016'}
{attribute addProperty BoxType "EP1258-0001-0016"}
{attribute addProperty Id "WcState0AT %I*BOOL1WcState1AT %I*BOOL1InputToggle0AT %I*BOOL1InputToggle1AT %I*BOOL1"}
{attribute addProperty CRC "3038159460"}
{attribute addProperty Size "4"}
TYPE WcState_B516A264 EXTENDS InputBase_8311D824 :
STRUCT
	{attribute addProperty Name "WcState0"}
	WcState0 AT %I* : BOOL;
	{attribute addProperty Name "WcState1"}
	WcState1 AT %I* : BOOL;
	{attribute addProperty Name "InputToggle0"}
	InputToggle0 AT %I* : BOOL;
	{attribute addProperty Name "InputToggle1"}
	InputToggle1 AT %I* : BOOL;
END_STRUCT
END_TYPE

// ---- DUTs/IO/PDOs/InfoData_A7436BC6.TcDUT
{attribute 'GeneratedUsingTerminal: EP1258-0001-0016'}
{attribute addProperty BoxType "EP1258-0001-0016"}
{attribute addProperty Id "DcOutputShiftAT %I*DINT4DcInputShiftAT %I*DINT4StateAT %I*UINT2"}
{attribute addProperty CRC "2806213574"}
{attribute addProperty Size "10"}
TYPE InfoData_A7436BC6 EXTENDS InputBase_8311D824 :
STRUCT
	{attribute addProperty Name "DcOutputShift"}
	DcOutputShift AT %I* : DINT;
	{attribute addProperty Name "DcInputShift"}
	DcInputShift AT %I* : DINT;
	{attribute addProperty Name "State"}
	State AT %I* : UINT;
END_STRUCT
END_TYPE

// ---- DUTs/IO/PDOs/CNT_Input_Channel_FF10BD3C.TcDUT
{attribute 'GeneratedUsingTerminal: EP1518-0002-0016'}
{attribute addProperty BoxType "EP1518-0002-0016"}
{attribute addProperty Id "StatusAT %I*Status_57491DF17Counter_valueAT %I*UDINT4"}
{attribute addProperty CRC "4279287100"}
{attribute addProperty Size "11"}
TYPE CNT_Input_Channel_FF10BD3C EXTENDS InputBase_8311D824 :
STRUCT
	{attribute addProperty Name "Status"}
	Status AT %I* : Status_57491DF1;
	{attribute addProperty Name "Counter_value"}
	Counter_value AT %I* : UDINT;
END_STRUCT
END_TYPE

// ---- DUTs/IO/PDOs/DIG_Inputs_CAFF6004.TcDUT
{attribute 'GeneratedUsingTerminal: EP1518-0002-0016'}
{attribute addProperty BoxType "EP1518-0002-0016"}
{attribute addProperty Id "InputAT %I*ARRAY[0..7] OF BOOL8"}
{attribute addProperty CRC "3697175534"}
{attribute addProperty Size "8"}
TYPE DIG_Inputs_CAFF6004 EXTENDS InputBase_8311D824 :
STRUCT
	{attribute addProperty Name "Input"}
	Input AT %I* : ARRAY[0..7] OF BOOL;
END_STRUCT
END_TYPE

// ---- DUTs/IO/PDOs/DIG_Inputs_Device_1F4E72EB.TcDUT
{attribute 'GeneratedUsingTerminal: EP1518-0002-0016'}
{attribute addProperty BoxType "EP1518-0002-0016"}
{attribute addProperty Id "StatusAT %I*Status_D4FDECD45"}
{attribute addProperty CRC "525234923"}
{attribute addProperty Size "5"}
TYPE DIG_Inputs_Device_1F4E72EB EXTENDS InputBase_8311D824 :
STRUCT
	{attribute addProperty Name "Status"}
	Status AT %I* : Status_D4FDECD4;
END_STRUCT
END_TYPE

// ---- DUTs/IO/PDOs/CNT_Output_Channel_550BB6DF.TcDUT
{attribute 'GeneratedUsingTerminal: EP1518-0002-0016'}
{attribute addProperty BoxType "EP1518-0002-0016"}
{attribute addProperty Id "ControlAT %Q*Control_0B2F8B702Set_counter_valueAT %Q*UDINT4"}
{attribute addProperty CRC "1426831071"}
{attribute addProperty Size "6"}
TYPE CNT_Output_Channel_550BB6DF EXTENDS OutputBase_10CEE7DE :
STRUCT
	{attribute addProperty Name "Control"}
	Control AT %Q* : Control_0B2F8B70;
	{attribute addProperty Name "Set_counter_value"}
	Set_counter_value AT %Q* : UDINT;
END_STRUCT
END_TYPE

// ---- DUTs/IO/PDOs/DI_X01_Pin_830843C1.TcDUT
{attribute 'GeneratedUsingTerminal: EP1809-0042-0018'}
{attribute addProperty BoxType "EP1809-0042-0018"}
{attribute addProperty Id "InputAT %I*BOOL1"}
{attribute addProperty CRC "2198356929"}
{attribute addProperty Size "1"}
TYPE DI_X01_Pin_830843C1 EXTENDS InputBase_8311D824 :
STRUCT
	{attribute addProperty Name "Input"}
	Input AT %I* : BOOL;
END_STRUCT
END_TYPE

// ---- DUTs/IO/PDOs/DI_X02_Pin_830843C1.TcDUT
{attribute 'GeneratedUsingTerminal: EP1809-0042-0018'}
{attribute addProperty BoxType "EP1809-0042-0018"}
{attribute addProperty Id "InputAT %I*BOOL1"}
{attribute addProperty CRC "2198356929"}
{attribute addProperty Size "1"}
TYPE DI_X02_Pin_830843C1 EXTENDS InputBase_8311D824 :
STRUCT
	{attribute addProperty Name "Input"}
	Input AT %I* : BOOL;
END_STRUCT
END_TYPE

// ---- DUTs/IO/PDOs/DI_X03_Pin_830843C1.TcDUT
{attribute 'GeneratedUsingTerminal: EP1809-0042-0018'}
{attribute addProperty BoxType "EP1809-0042-0018"}
{attribute addProperty Id "InputAT %I*BOOL1"}
{attribute addProperty CRC "2198356929"}
{attribute addProperty Size "1"}
TYPE DI_X03_Pin_830843C1 EXTENDS InputBase_8311D824 :
STRUCT
	{attribute addProperty Name "Input"}
	Input AT %I* : BOOL;
END_STRUCT
END_TYPE

// ---- DUTs/IO/PDOs/DI_X04_Pin_830843C1.TcDUT
{attribute 'GeneratedUsingTerminal: EP1809-0042-0018'}
{attribute addProperty BoxType "EP1809-0042-0018"}
{attribute addProperty Id "InputAT %I*BOOL1"}
{attribute addProperty CRC "2198356929"}
{attribute addProperty Size "1"}
TYPE DI_X04_Pin_830843C1 EXTENDS InputBase_8311D824 :
STRUCT
	{attribute addProperty Name "Input"}
	Input AT %I* : BOOL;
END_STRUCT
END_TYPE

// ---- DUTs/IO/PDOs/DI_X05_Pin_830843C1.TcDUT
{attribute 'GeneratedUsingTerminal: EP1809-0042-0018'}
{attribute addProperty BoxType "EP1809-0042-0018"}
{attribute addProperty Id "InputAT %I*BOOL1"}
{attribute addProperty CRC "2198356929"}
{attribute addProperty Size "1"}
TYPE DI_X05_Pin_830843C1 EXTENDS InputBase_8311D824 :
STRUCT
	{attribute addProperty Name "Input"}
	Input AT %I* : BOOL;
END_STRUCT
END_TYPE

// ---- DUTs/IO/PDOs/DI_X06_Pin_830843C1.TcDUT
{attribute 'GeneratedUsingTerminal: EP1809-0042-0018'}
{attribute addProperty BoxType "EP1809-0042-0018"}
{attribute addProperty Id "InputAT %I*BOOL1"}
{attribute addProperty CRC "2198356929"}
{attribute addProperty Size "1"}
TYPE DI_X06_Pin_830843C1 EXTENDS InputBase_8311D824 :
STRUCT
	{attribute addProperty Name "Input"}
	Input AT %I* : BOOL;
END_STRUCT
END_TYPE

// ---- DUTs/IO/PDOs/DI_X07_Pin_830843C1.TcDUT
{attribute 'GeneratedUsingTerminal: EP1809-0042-0018'}
{attribute addProperty BoxType "EP1809-0042-0018"}
{attribute addProperty Id "InputAT %I*BOOL1"}
{attribute addProperty CRC "2198356929"}
{attribute addProperty Size "1"}
TYPE DI_X07_Pin_830843C1 EXTENDS InputBase_8311D824 :
STRUCT
	{attribute addProperty Name "Input"}
	Input AT %I* : BOOL;
END_STRUCT
END_TYPE

// ---- DUTs/IO/PDOs/DI_X08_Pin_830843C1.TcDUT
{attribute 'GeneratedUsingTerminal: EP1809-0042-0018'}
{attribute addProperty BoxType "EP1809-0042-0018"}
{attribute addProperty Id "InputAT %I*BOOL1"}
{attribute addProperty CRC "2198356929"}
{attribute addProperty Size "1"}
TYPE DI_X08_Pin_830843C1 EXTENDS InputBase_8311D824 :
STRUCT
	{attribute addProperty Name "Input"}
	Input AT %I* : BOOL;
END_STRUCT
END_TYPE

// ---- DUTs/IO/PDOs/DI_X_830843C1.TcDUT
{attribute 'GeneratedUsingTerminal: EP1809-0042-0019'}
{attribute addProperty BoxType "EP1809-0042-0019"}
{attribute addProperty Id "InputAT %I*BOOL1"}
{attribute addProperty CRC "2198356929"}
{attribute addProperty Size "1"}
TYPE DI_X_830843C1 EXTENDS InputBase_8311D824 :
STRUCT
	{attribute addProperty Name "Input"}
	Input AT %I* : BOOL;
END_STRUCT
END_TYPE

// ---- DUTs/IO/PDOs/DIG_Inputs_Channel_ACAA0425.TcDUT
{attribute 'GeneratedUsingTerminal: EP1816-0003-0016'}
{attribute addProperty BoxType "EP1816-0003-0016"}
{attribute addProperty Id "InputAT %I*ARRAY[0..7] OF BOOL8Sync_errorAT %I*BOOL1TxPDO_ToggleAT %I*BOOL1"}
{attribute addProperty CRC "780220065"}
{attribute addProperty Size "10"}
TYPE DIG_Inputs_Channel_ACAA0425 EXTENDS InputBase_8311D824 :
STRUCT
	{attribute addProperty Name "Input"}
	Input AT %I* : ARRAY[0..7] OF BOOL;
	{attribute addProperty Name "Sync_error"}
	Sync_error AT %I* : BOOL;
	{attribute addProperty Name "TxPDO_Toggle"}
	TxPDO_Toggle AT %I* : BOOL;
END_STRUCT
END_TYPE

// ---- DUTs/IO/PDOs/DO_Inputs_Channel_CC455148.TcDUT
{attribute 'GeneratedUsingTerminal: EP1816-0008-0016'}
{attribute addProperty BoxType "EP1816-0008-0016"}
{attribute addProperty Id "InputAT %I*ARRAY[0..7] OF BOOL8Sync_ErrorAT %I*BOOL1"}
{attribute addProperty CRC "2788215981"}
{attribute addProperty Size "9"}
TYPE DO_Inputs_Channel_CC455148 EXTENDS InputBase_8311D824 :
STRUCT
	{attribute addProperty Name "Input"}
	Input AT %I* : ARRAY[0..7] OF BOOL;
	{attribute addProperty Name "Sync_Error"}
	Sync_Error AT %I* : BOOL;
END_STRUCT
END_TYPE

// ---- DUTs/IO/PDOs/DIG_Inputs_Channel_CC455148.TcDUT
{attribute 'GeneratedUsingTerminal: EP1816-0008-0018'}
{attribute addProperty BoxType "EP1816-0008-0018"}
{attribute addProperty Id "InputAT %I*ARRAY[0..7] OF BOOL8Sync_ErrorAT %I*BOOL1"}
{attribute addProperty CRC "2788215981"}
{attribute addProperty Size "9"}
TYPE DIG_Inputs_Channel_CC455148 EXTENDS InputBase_8311D824 :
STRUCT
	{attribute addProperty Name "Input"}
	Input AT %I* : ARRAY[0..7] OF BOOL;
	{attribute addProperty Name "Sync_Error"}
	Sync_Error AT %I* : BOOL;
END_STRUCT
END_TYPE

// ---- DUTs/IO/PDOs/DIG_Inputs_Channel_38F9DD27.TcDUT
{attribute 'GeneratedUsingTerminal: EP1816-1008-0016'}
{attribute addProperty BoxType "EP1816-1008-0016"}
{attribute addProperty Id "InputAT %I*ARRAY[0..7] OF BOOL8"}
{attribute addProperty CRC "3697175534"}
{attribute addProperty Size "8"}
TYPE DIG_Inputs_Channel_38F9DD27 EXTENDS InputBase_8311D824 :
STRUCT
	{attribute addProperty Name "Input"}
	Input AT %I* : ARRAY[0..7] OF BOOL;
END_STRUCT
END_TYPE

// ---- DUTs/IO/PDOs/DIG_Inputs_Device_B3EA4204.TcDUT
{attribute 'GeneratedUsingTerminal: EP1816-1008-0016'}
{attribute addProperty BoxType "EP1816-1008-0016"}
{attribute addProperty Id "Us_UndervoltageAT %I*BOOL1Up_UndervoltageAT %I*BOOL1Sync_errorAT %I*BOOL1TxPDO_ToggleAT %I*BOOL1"}
{attribute addProperty CRC "3018473988"}
{attribute addProperty Size "4"}
TYPE DIG_Inputs_Device_B3EA4204 EXTENDS InputBase_8311D824 :
STRUCT
	{attribute addProperty Name "Us_Undervoltage"}
	Us_Undervoltage AT %I* : BOOL;
	{attribute addProperty Name "Up_Undervoltage"}
	Up_Undervoltage AT %I* : BOOL;
	{attribute addProperty Name "Sync_error"}
	Sync_error AT %I* : BOOL;
	{attribute addProperty Name "TxPDO_Toggle"}
	TxPDO_Toggle AT %I* : BOOL;
END_STRUCT
END_TYPE

// ---- DUTs/IO/PDOs/AI_Inputs_Channel_C3DE7A0A.TcDUT
{attribute 'GeneratedUsingTerminal: EP1816-3008-0016'}
{attribute addProperty BoxType "EP1816-3008-0016"}
{attribute addProperty Id "StatusAT %I*Status_A3AA621F2ValueAT %I*INT2"}
{attribute addProperty CRC "3286137354"}
{attribute addProperty Size "4"}
TYPE AI_Inputs_Channel_C3DE7A0A EXTENDS InputBase_8311D824 :
STRUCT
	{attribute addProperty Name "Status"}
	Status AT %I* : Status_A3AA621F;
	{attribute addProperty Name "Value"}
	Value AT %I* : INT;
END_STRUCT
END_TYPE

// ---- DUTs/IO/PDOs/DO_X05_Pin_42CA91F7.TcDUT
{attribute 'GeneratedUsingTerminal: EP1859-0042-0018'}
{attribute addProperty BoxType "EP1859-0042-0018"}
{attribute addProperty Id "OutputAT %Q*BOOL1"}
{attribute addProperty CRC "1120571895"}
{attribute addProperty Size "1"}
TYPE DO_X05_Pin_42CA91F7 EXTENDS OutputBase_10CEE7DE :
STRUCT
	{attribute addProperty Name "Output"}
	Output AT %Q* : BOOL;
END_STRUCT
END_TYPE

// ---- DUTs/IO/PDOs/DO_X06_Pin_42CA91F7.TcDUT
{attribute 'GeneratedUsingTerminal: EP1859-0042-0018'}
{attribute addProperty BoxType "EP1859-0042-0018"}
{attribute addProperty Id "OutputAT %Q*BOOL1"}
{attribute addProperty CRC "1120571895"}
{attribute addProperty Size "1"}
TYPE DO_X06_Pin_42CA91F7 EXTENDS OutputBase_10CEE7DE :
STRUCT
	{attribute addProperty Name "Output"}
	Output AT %Q* : BOOL;
END_STRUCT
END_TYPE

// ---- DUTs/IO/PDOs/DO_X07_Pin_42CA91F7.TcDUT
{attribute 'GeneratedUsingTerminal: EP1859-0042-0018'}
{attribute addProperty BoxType "EP1859-0042-0018"}
{attribute addProperty Id "OutputAT %Q*BOOL1"}
{attribute addProperty CRC "1120571895"}
{attribute addProperty Size "1"}
TYPE DO_X07_Pin_42CA91F7 EXTENDS OutputBase_10CEE7DE :
STRUCT
	{attribute addProperty Name "Output"}
	Output AT %Q* : BOOL;
END_STRUCT
END_TYPE

// ---- DUTs/IO/PDOs/DO_X08_Pin_42CA91F7.TcDUT
{attribute 'GeneratedUsingTerminal: EP1859-0042-0018'}
{attribute addProperty BoxType "EP1859-0042-0018"}
{attribute addProperty Id "OutputAT %Q*BOOL1"}
{attribute addProperty CRC "1120571895"}
{attribute addProperty Size "1"}
TYPE DO_X08_Pin_42CA91F7 EXTENDS OutputBase_10CEE7DE :
STRUCT
	{attribute addProperty Name "Output"}
	Output AT %Q* : BOOL;
END_STRUCT
END_TYPE

// ---- DUTs/IO/PDOs/DO_X_42CA91F7.TcDUT
{attribute 'GeneratedUsingTerminal: EP1859-0042-0019'}
{attribute addProperty BoxType "EP1859-0042-0019"}
{attribute addProperty Id "OutputAT %Q*BOOL1"}
{attribute addProperty CRC "1120571895"}
{attribute addProperty Size "1"}
TYPE DO_X_42CA91F7 EXTENDS OutputBase_10CEE7DE :
STRUCT
	{attribute addProperty Name "Output"}
	Output AT %Q* : BOOL;
END_STRUCT
END_TYPE

// ---- DUTs/IO/PDOs/Group_99EF3D30.TcDUT
{attribute 'GeneratedUsingTerminal: EP2001-1000-0016'}
{attribute addProperty BoxType "EP2001-1000-0016"}
{attribute addProperty Id "Output1AT %Q*BOOL1Output2AT %Q*BOOL1Output3AT %Q*BOOL1Output4AT %Q*BOOL1"}
{attribute addProperty CRC "2582592816"}
{attribute addProperty Size "4"}
TYPE Group_99EF3D30 EXTENDS OutputBase_10CEE7DE :
STRUCT
	{attribute addProperty Name "Output1"}
	Output1 AT %Q* : BOOL;
	{attribute addProperty Name "Output2"}
	Output2 AT %Q* : BOOL;
	{attribute addProperty Name "Output3"}
	Output3 AT %Q* : BOOL;
	{attribute addProperty Name "Output4"}
	Output4 AT %Q* : BOOL;
END_STRUCT
END_TYPE

// ---- DUTs/IO/PDOs/Group_8FCDB395.TcDUT
{attribute 'GeneratedUsingTerminal: EP2001-1000-0016'}
{attribute addProperty BoxType "EP2001-1000-0016"}
{attribute addProperty Id "Output5AT %Q*BOOL1Output6AT %Q*BOOL1Output7AT %Q*BOOL1Output8AT %Q*BOOL1"}
{attribute addProperty CRC "2412622741"}
{attribute addProperty Size "4"}
TYPE Group_8FCDB395 EXTENDS OutputBase_10CEE7DE :
STRUCT
	{attribute addProperty Name "Output5"}
	Output5 AT %Q* : BOOL;
	{attribute addProperty Name "Output6"}
	Output6 AT %Q* : BOOL;
	{attribute addProperty Name "Output7"}
	Output7 AT %Q* : BOOL;
	{attribute addProperty Name "Output8"}
	Output8 AT %Q* : BOOL;
END_STRUCT
END_TYPE

// ---- DUTs/IO/PDOs/WcState_0B2B16F9.TcDUT
{attribute 'GeneratedUsingTerminal: EP2001-1000-0016'}
{attribute addProperty BoxType "EP2001-1000-0016"}
{attribute addProperty Id "WcStateAT %I*BOOL1"}
{attribute addProperty CRC "187373305"}
{attribute addProperty Size "1"}
TYPE WcState_0B2B16F9 :
STRUCT
	{attribute addProperty Name "WcState"}
	WcState AT %I* : BOOL;
END_STRUCT
END_TYPE

// ---- DUTs/IO/PDOs/Channel_42CA91F7.TcDUT
{attribute 'GeneratedUsingTerminal: EP2008-0001-0016'}
{attribute addProperty BoxType "EP2008-0001-0016"}
{attribute addProperty Id "OutputAT %Q*BOOL1"}
{attribute addProperty CRC "1120571895"}
{attribute addProperty Size "1"}
TYPE Channel_42CA91F7 EXTENDS OutputBase_10CEE7DE :
STRUCT
	{attribute addProperty Name "Output"}
	Output AT %Q* : BOOL;
END_STRUCT
END_TYPE

// ---- DUTs/IO/PDOs/Diag_Channel_830843C1.TcDUT
{attribute 'GeneratedUsingTerminal: EP2038-0001-0016'}
{attribute addProperty BoxType "EP2038-0001-0016"}
{attribute addProperty Id "InputAT %I*BOOL1"}
{attribute addProperty CRC "2198356929"}
{attribute addProperty Size "1"}
TYPE Diag_Channel_830843C1 EXTENDS InputBase_8311D824 :
STRUCT
	{attribute addProperty Name "Input"}
	Input AT %I* : BOOL;
END_STRUCT
END_TYPE

// ---- DUTs/IO/PDOs/DIG_Inputs_CC455148.TcDUT
{attribute 'GeneratedUsingTerminal: EP2316-0003-0016'}
{attribute addProperty BoxType "EP2316-0003-0016"}
{attribute addProperty Id "InputAT %I*ARRAY[0..7] OF BOOL8Sync_ErrorAT %I*BOOL1"}
{attribute addProperty CRC "2788215981"}
{attribute addProperty Size "9"}
TYPE DIG_Inputs_CC455148 EXTENDS InputBase_8311D824 :
STRUCT
	{attribute addProperty Name "Input"}
	Input AT %I* : ARRAY[0..7] OF BOOL;
	{attribute addProperty Name "Sync_Error"}
	Sync_Error AT %I* : BOOL;
END_STRUCT
END_TYPE

// ---- DUTs/IO/PDOs/DIG_Diag_Inputs_584303BF.TcDUT
{attribute 'GeneratedUsingTerminal: EP2316-0003-0016'}
{attribute addProperty BoxType "EP2316-0003-0016"}
{attribute addProperty Id "Diag_InputAT %I*ARRAY[0..7] OF BOOL8"}
{attribute addProperty CRC "568896300"}
{attribute addProperty Size "8"}
TYPE DIG_Diag_Inputs_584303BF EXTENDS InputBase_8311D824 :
STRUCT
	{attribute addProperty Name "Diag_Input"}
	Diag_Input AT %I* : ARRAY[0..7] OF BOOL;
END_STRUCT
END_TYPE

// ---- DUTs/IO/PDOs/DIG_Inputs_Device_E94E5BF9.TcDUT
{attribute 'GeneratedUsingTerminal: EP2316-0003-0016'}
{attribute addProperty BoxType "EP2316-0003-0016"}
{attribute addProperty Id "Safe_state_activeAT %I*BOOL1Error_channelAT %I*ARRAY[0..1] OF BOOL2Sync_errorAT %I*BOOL1TxPDO_ToggleAT %I*BOOL1"}
{attribute addProperty CRC "304706677"}
{attribute addProperty Size "5"}
TYPE DIG_Inputs_Device_E94E5BF9 EXTENDS InputBase_8311D824 :
STRUCT
	{attribute addProperty Name "Safe_state_active"}
	Safe_state_active AT %I* : BOOL;
	{attribute addProperty Name "Error_channel"}
	Error_channel AT %I* : ARRAY[0..1] OF BOOL;
	{attribute addProperty Name "Sync_error"}
	Sync_error AT %I* : BOOL;
	{attribute addProperty Name "TxPDO_Toggle"}
	TxPDO_Toggle AT %I* : BOOL;
END_STRUCT
END_TYPE

// ---- DUTs/IO/PDOs/DIG_Outputs_28AC1A9E.TcDUT
{attribute 'GeneratedUsingTerminal: EP2316-0003-0016'}
{attribute addProperty BoxType "EP2316-0003-0016"}
{attribute addProperty Id "OutputAT %Q*ARRAY[0..7] OF BOOL8"}
{attribute addProperty CRC "1253840710"}
{attribute addProperty Size "8"}
TYPE DIG_Outputs_28AC1A9E EXTENDS OutputBase_10CEE7DE :
STRUCT
	{attribute addProperty Name "Output"}
	Output AT %Q* : ARRAY[0..7] OF BOOL;
END_STRUCT
END_TYPE

// ---- DUTs/IO/PDOs/DIG_Outputs_Device_36A5EF17.TcDUT
{attribute 'GeneratedUsingTerminal: EP2316-0003-0016'}
{attribute addProperty BoxType "EP2316-0003-0016"}
{attribute addProperty Id "Set_safe_stateAT %Q*BOOL1Reset_outputsAT %Q*BOOL1"}
{attribute addProperty CRC "916844311"}
{attribute addProperty Size "2"}
TYPE DIG_Outputs_Device_36A5EF17 EXTENDS OutputBase_10CEE7DE :
STRUCT
	{attribute addProperty Name "Set_safe_state"}
	Set_safe_state AT %Q* : BOOL;
	{attribute addProperty Name "Reset_outputs"}
	Reset_outputs AT %Q* : BOOL;
END_STRUCT
END_TYPE

// ---- DUTs/IO/PDOs/DO_Inputs_CC455148.TcDUT
{attribute 'GeneratedUsingTerminal: EP2316-0008-0016'}
{attribute addProperty BoxType "EP2316-0008-0016"}
{attribute addProperty Id "InputAT %I*ARRAY[0..7] OF BOOL8Sync_ErrorAT %I*BOOL1"}
{attribute addProperty CRC "2788215981"}
{attribute addProperty Size "9"}
TYPE DO_Inputs_CC455148 EXTENDS InputBase_8311D824 :
STRUCT
	{attribute addProperty Name "Input"}
	Input AT %I* : ARRAY[0..7] OF BOOL;
	{attribute addProperty Name "Sync_Error"}
	Sync_Error AT %I* : BOOL;
END_STRUCT
END_TYPE

// ---- DUTs/IO/PDOs/DO_Diag_Inputs_584303BF.TcDUT
{attribute 'GeneratedUsingTerminal: EP2316-0008-0016'}
{attribute addProperty BoxType "EP2316-0008-0016"}
{attribute addProperty Id "Diag_InputAT %I*ARRAY[0..7] OF BOOL8"}
{attribute addProperty CRC "568896300"}
{attribute addProperty Size "8"}
TYPE DO_Diag_Inputs_584303BF EXTENDS InputBase_8311D824 :
STRUCT
	{attribute addProperty Name "Diag_Input"}
	Diag_Input AT %I* : ARRAY[0..7] OF BOOL;
END_STRUCT
END_TYPE

// ---- DUTs/IO/PDOs/DO_Inputs_Device_AF161A9E.TcDUT
{attribute 'GeneratedUsingTerminal: EP2316-0008-0016'}
{attribute addProperty BoxType "EP2316-0008-0016"}
{attribute addProperty Id "Safe_state_activeAT %I*BOOL1Error_channel_1AT %I*BOOL1Sync_ErrorAT %I*BOOL1TxPDO_ToggleAT %I*BOOL1"}
{attribute addProperty CRC "2937461406"}
{attribute addProperty Size "4"}
TYPE DO_Inputs_Device_AF161A9E EXTENDS InputBase_8311D824 :
STRUCT
	{attribute addProperty Name "Safe_state_active"}
	Safe_state_active AT %I* : BOOL;
	{attribute addProperty Name "Error_channel_1"}
	Error_channel_1 AT %I* : BOOL;
	{attribute addProperty Name "Sync_Error"}
	Sync_Error AT %I* : BOOL;
	{attribute addProperty Name "TxPDO_Toggle"}
	TxPDO_Toggle AT %I* : BOOL;
END_STRUCT
END_TYPE

// ---- DUTs/IO/PDOs/DO_Outputs_28AC1A9E.TcDUT
{attribute 'GeneratedUsingTerminal: EP2316-0008-0016'}
{attribute addProperty BoxType "EP2316-0008-0016"}
{attribute addProperty Id "OutputAT %Q*ARRAY[0..7] OF BOOL8"}
{attribute addProperty CRC "1253840710"}
{attribute addProperty Size "8"}
TYPE DO_Outputs_28AC1A9E EXTENDS OutputBase_10CEE7DE :
STRUCT
	{attribute addProperty Name "Output"}
	Output AT %Q* : ARRAY[0..7] OF BOOL;
END_STRUCT
END_TYPE

// ---- DUTs/IO/PDOs/DO_Outputs_Device_36A5EF17.TcDUT
{attribute 'GeneratedUsingTerminal: EP2316-0008-0016'}
{attribute addProperty BoxType "EP2316-0008-0016"}
{attribute addProperty Id "Set_safe_stateAT %Q*BOOL1Reset_outputsAT %Q*BOOL1"}
{attribute addProperty CRC "916844311"}
{attribute addProperty Size "2"}
TYPE DO_Outputs_Device_36A5EF17 EXTENDS OutputBase_10CEE7DE :
STRUCT
	{attribute addProperty Name "Set_safe_state"}
	Set_safe_state AT %Q* : BOOL;
	{attribute addProperty Name "Reset_outputs"}
	Reset_outputs AT %Q* : BOOL;
END_STRUCT
END_TYPE

// ---- DUTs/IO/PDOs/DO_Diag_Inputs_CC455148.TcDUT
{attribute 'GeneratedUsingTerminal: EP2316-0008-0017'}
{attribute addProperty BoxType "EP2316-0008-0017"}
{attribute addProperty Id "InputAT %I*ARRAY[0..7] OF BOOL8Sync_ErrorAT %I*BOOL1"}
{attribute addProperty CRC "2788215981"}
{attribute addProperty Size "9"}
TYPE DO_Diag_Inputs_CC455148 EXTENDS InputBase_8311D824 :
STRUCT
	{attribute addProperty Name "Input"}
	Input AT %I* : ARRAY[0..7] OF BOOL;
	{attribute addProperty Name "Sync_Error"}
	Sync_Error AT %I* : BOOL;
END_STRUCT
END_TYPE

// ---- DUTs/IO/PDOs/DO_Diag_Inputs_212B82C1.TcDUT
{attribute 'GeneratedUsingTerminal: EP2316-0008-0017'}
{attribute addProperty BoxType "EP2316-0008-0017"}
{attribute addProperty Id "Diag_InputAT %I*ARRAY[0..7] OF BOOL8Sync_ErrorAT %I*BOOL1"}
{attribute addProperty CRC "3811544510"}
{attribute addProperty Size "9"}
TYPE DO_Diag_Inputs_212B82C1 EXTENDS InputBase_8311D824 :
STRUCT
	{attribute addProperty Name "Diag_Input"}
	Diag_Input AT %I* : ARRAY[0..7] OF BOOL;
	{attribute addProperty Name "Sync_Error"}
	Sync_Error AT %I* : BOOL;
END_STRUCT
END_TYPE

// ---- DUTs/IO/PDOs/DIG_Inputs_Device_4E5AF17E.TcDUT
{attribute 'GeneratedUsingTerminal: EP2316-0008-0018'}
{attribute addProperty BoxType "EP2316-0008-0018"}
{attribute addProperty Id "Safe_state_activeAT %I*BOOL1Error_channelAT %I*ARRAY[0..1] OF BOOL2Sync_ErrorAT %I*BOOL1TxPDO_ToggleAT %I*BOOL1"}
{attribute addProperty CRC "3040730866"}
{attribute addProperty Size "5"}
TYPE DIG_Inputs_Device_4E5AF17E EXTENDS InputBase_8311D824 :
STRUCT
	{attribute addProperty Name "Safe_state_active"}
	Safe_state_active AT %I* : BOOL;
	{attribute addProperty Name "Error_channel"}
	Error_channel AT %I* : ARRAY[0..1] OF BOOL;
	{attribute addProperty Name "Sync_Error"}
	Sync_Error AT %I* : BOOL;
	{attribute addProperty Name "TxPDO_Toggle"}
	TxPDO_Toggle AT %I* : BOOL;
END_STRUCT
END_TYPE

// ---- DUTs/IO/PDOs/DI_X01_Pin4_Input_830843C1.TcDUT
{attribute 'GeneratedUsingTerminal: EP2328-1061-0016'}
{attribute addProperty BoxType "EP2328-1061-0016"}
{attribute addProperty Id "InputAT %I*BOOL1"}
{attribute addProperty CRC "2198356929"}
{attribute addProperty Size "1"}
TYPE DI_X01_Pin4_Input_830843C1 EXTENDS InputBase_8311D824 :
STRUCT
	{attribute addProperty Name "Input"}
	Input AT %I* : BOOL;
END_STRUCT
END_TYPE

// ---- DUTs/IO/PDOs/DI_X01_Pin2_Input_830843C1.TcDUT
{attribute 'GeneratedUsingTerminal: EP2328-1061-0016'}
{attribute addProperty BoxType "EP2328-1061-0016"}
{attribute addProperty Id "InputAT %I*BOOL1"}
{attribute addProperty CRC "2198356929"}
{attribute addProperty Size "1"}
TYPE DI_X01_Pin2_Input_830843C1 EXTENDS InputBase_8311D824 :
STRUCT
	{attribute addProperty Name "Input"}
	Input AT %I* : BOOL;
END_STRUCT
END_TYPE

// ---- DUTs/IO/PDOs/DI_X02_Pin4_Input_830843C1.TcDUT
{attribute 'GeneratedUsingTerminal: EP2328-1061-0016'}
{attribute addProperty BoxType "EP2328-1061-0016"}
{attribute addProperty Id "InputAT %I*BOOL1"}
{attribute addProperty CRC "2198356929"}
{attribute addProperty Size "1"}
TYPE DI_X02_Pin4_Input_830843C1 EXTENDS InputBase_8311D824 :
STRUCT
	{attribute addProperty Name "Input"}
	Input AT %I* : BOOL;
END_STRUCT
END_TYPE

// ---- DUTs/IO/PDOs/DI_X02_Pin2_Input_830843C1.TcDUT
{attribute 'GeneratedUsingTerminal: EP2328-1061-0016'}
{attribute addProperty BoxType "EP2328-1061-0016"}
{attribute addProperty Id "InputAT %I*BOOL1"}
{attribute addProperty CRC "2198356929"}
{attribute addProperty Size "1"}
TYPE DI_X02_Pin2_Input_830843C1 EXTENDS InputBase_8311D824 :
STRUCT
	{attribute addProperty Name "Input"}
	Input AT %I* : BOOL;
END_STRUCT
END_TYPE

// ---- DUTs/IO/PDOs/DO_X03_Pin4_Output_42CA91F7.TcDUT
{attribute 'GeneratedUsingTerminal: EP2328-1061-0016'}
{attribute addProperty BoxType "EP2328-1061-0016"}
{attribute addProperty Id "OutputAT %Q*BOOL1"}
{attribute addProperty CRC "1120571895"}
{attribute addProperty Size "1"}
TYPE DO_X03_Pin4_Output_42CA91F7 EXTENDS OutputBase_10CEE7DE :
STRUCT
	{attribute addProperty Name "Output"}
	Output AT %Q* : BOOL;
END_STRUCT
END_TYPE

// ---- DUTs/IO/PDOs/DO_X03_Pin2_Output_42CA91F7.TcDUT
{attribute 'GeneratedUsingTerminal: EP2328-1061-0016'}
{attribute addProperty BoxType "EP2328-1061-0016"}
{attribute addProperty Id "OutputAT %Q*BOOL1"}
{attribute addProperty CRC "1120571895"}
{attribute addProperty Size "1"}
TYPE DO_X03_Pin2_Output_42CA91F7 EXTENDS OutputBase_10CEE7DE :
STRUCT
	{attribute addProperty Name "Output"}
	Output AT %Q* : BOOL;
END_STRUCT
END_TYPE

// ---- DUTs/IO/PDOs/DO_X04_Pin4_Output_42CA91F7.TcDUT
{attribute 'GeneratedUsingTerminal: EP2328-1061-0016'}
{attribute addProperty BoxType "EP2328-1061-0016"}
{attribute addProperty Id "OutputAT %Q*BOOL1"}
{attribute addProperty CRC "1120571895"}
{attribute addProperty Size "1"}
TYPE DO_X04_Pin4_Output_42CA91F7 EXTENDS OutputBase_10CEE7DE :
STRUCT
	{attribute addProperty Name "Output"}
	Output AT %Q* : BOOL;
END_STRUCT
END_TYPE

// ---- DUTs/IO/PDOs/DO_X04_Pin2_Output_42CA91F7.TcDUT
{attribute 'GeneratedUsingTerminal: EP2328-1061-0016'}
{attribute addProperty BoxType "EP2328-1061-0016"}
{attribute addProperty Id "OutputAT %Q*BOOL1"}
{attribute addProperty CRC "1120571895"}
{attribute addProperty Size "1"}
TYPE DO_X04_Pin2_Output_42CA91F7 EXTENDS OutputBase_10CEE7DE :
STRUCT
	{attribute addProperty Name "Output"}
	Output AT %Q* : BOOL;
END_STRUCT
END_TYPE

// ---- DUTs/IO/PDOs/DI_Inputs_Channel_91AC31B7.TcDUT
{attribute 'GeneratedUsingTerminal: EP2339-0003-0016'}
{attribute addProperty BoxType "EP2339-0003-0016"}
{attribute addProperty Id "InputAT %I*ARRAY[0..7] OF BOOL8Sync_errorAT %I*BOOL1TxPDO_StateAT %I*BOOL1TxPDO_ToggleAT %I*BOOL1"}
{attribute addProperty CRC "1559998493"}
{attribute addProperty Size "11"}
TYPE DI_Inputs_Channel_91AC31B7 EXTENDS InputBase_8311D824 :
STRUCT
	{attribute addProperty Name "Input"}
	Input AT %I* : ARRAY[0..7] OF BOOL;
	{attribute addProperty Name "Sync_error"}
	Sync_error AT %I* : BOOL;
	{attribute addProperty Name "TxPDO_State"}
	TxPDO_State AT %I* : BOOL;
	{attribute addProperty Name "TxPDO_Toggle"}
	TxPDO_Toggle AT %I* : BOOL;
END_STRUCT
END_TYPE

// ---- DUTs/IO/PDOs/DO_Outputs_Channel_28AC1A9E.TcDUT
{attribute 'GeneratedUsingTerminal: EP2339-0003-0016'}
{attribute addProperty BoxType "EP2339-0003-0016"}
{attribute addProperty Id "OutputAT %Q*ARRAY[0..7] OF BOOL8"}
{attribute addProperty CRC "1253840710"}
{attribute addProperty Size "8"}
TYPE DO_Outputs_Channel_28AC1A9E EXTENDS OutputBase_10CEE7DE :
STRUCT
	{attribute addProperty Name "Output"}
	Output AT %Q* : ARRAY[0..7] OF BOOL;
END_STRUCT
END_TYPE

// ---- DUTs/IO/PDOs/InfoData_0A66F009.TcDUT
{attribute 'GeneratedUsingTerminal: EP2339-0021-0016'}
{attribute addProperty BoxType "EP2339-0021-0016"}
{attribute addProperty Id "AoeNetIdAT %I*AMSNETID6StateAT %I*UINT2"}
{attribute addProperty CRC "174518281"}
{attribute addProperty Size "8"}
TYPE InfoData_0A66F009 EXTENDS InputBase_8311D824 :
STRUCT
	{attribute addProperty Name "AoeNetId"}
	AoeNetId AT %I* : AMSNETID;
	{attribute addProperty Name "State"}
	State AT %I* : UINT;
END_STRUCT
END_TYPE

// ---- DUTs/IO/PDOs/DO_X01_Pin_42CA91F7.TcDUT
{attribute 'GeneratedUsingTerminal: EP2339-0042-0017'}
{attribute addProperty BoxType "EP2339-0042-0017"}
{attribute addProperty Id "OutputAT %Q*BOOL1"}
{attribute addProperty CRC "1120571895"}
{attribute addProperty Size "1"}
TYPE DO_X01_Pin_42CA91F7 EXTENDS OutputBase_10CEE7DE :
STRUCT
	{attribute addProperty Name "Output"}
	Output AT %Q* : BOOL;
END_STRUCT
END_TYPE

// ---- DUTs/IO/PDOs/DO_X02_Pin_42CA91F7.TcDUT
{attribute 'GeneratedUsingTerminal: EP2339-0042-0017'}
{attribute addProperty BoxType "EP2339-0042-0017"}
{attribute addProperty Id "OutputAT %Q*BOOL1"}
{attribute addProperty CRC "1120571895"}
{attribute addProperty Size "1"}
TYPE DO_X02_Pin_42CA91F7 EXTENDS OutputBase_10CEE7DE :
STRUCT
	{attribute addProperty Name "Output"}
	Output AT %Q* : BOOL;
END_STRUCT
END_TYPE

// ---- DUTs/IO/PDOs/DO_X03_Pin_42CA91F7.TcDUT
{attribute 'GeneratedUsingTerminal: EP2339-0042-0017'}
{attribute addProperty BoxType "EP2339-0042-0017"}
{attribute addProperty Id "OutputAT %Q*BOOL1"}
{attribute addProperty CRC "1120571895"}
{attribute addProperty Size "1"}
TYPE DO_X03_Pin_42CA91F7 EXTENDS OutputBase_10CEE7DE :
STRUCT
	{attribute addProperty Name "Output"}
	Output AT %Q* : BOOL;
END_STRUCT
END_TYPE

// ---- DUTs/IO/PDOs/DO_X04_Pin_42CA91F7.TcDUT
{attribute 'GeneratedUsingTerminal: EP2339-0042-0017'}
{attribute addProperty BoxType "EP2339-0042-0017"}
{attribute addProperty Id "OutputAT %Q*BOOL1"}
{attribute addProperty CRC "1120571895"}
{attribute addProperty Size "1"}
TYPE DO_X04_Pin_42CA91F7 EXTENDS OutputBase_10CEE7DE :
STRUCT
	{attribute addProperty Name "Output"}
	Output AT %Q* : BOOL;
END_STRUCT
END_TYPE

// ---- DUTs/IO/PDOs/DIG_Diag_Inputs_Channel_584303BF.TcDUT
{attribute 'GeneratedUsingTerminal: EP2816-0003-0016'}
{attribute addProperty BoxType "EP2816-0003-0016"}
{attribute addProperty Id "Diag_InputAT %I*ARRAY[0..7] OF BOOL8"}
{attribute addProperty CRC "568896300"}
{attribute addProperty Size "8"}
TYPE DIG_Diag_Inputs_Channel_584303BF EXTENDS InputBase_8311D824 :
STRUCT
	{attribute addProperty Name "Diag_Input"}
	Diag_Input AT %I* : ARRAY[0..7] OF BOOL;
END_STRUCT
END_TYPE

// ---- DUTs/IO/PDOs/DIG_Output_Channel_28AC1A9E.TcDUT
{attribute 'GeneratedUsingTerminal: EP2816-0003-0016'}
{attribute addProperty BoxType "EP2816-0003-0016"}
{attribute addProperty Id "OutputAT %Q*ARRAY[0..7] OF BOOL8"}
{attribute addProperty CRC "1253840710"}
{attribute addProperty Size "8"}
TYPE DIG_Output_Channel_28AC1A9E EXTENDS OutputBase_10CEE7DE :
STRUCT
	{attribute addProperty Name "Output"}
	Output AT %Q* : ARRAY[0..7] OF BOOL;
END_STRUCT
END_TYPE

// ---- DUTs/IO/PDOs/DO_Inputs_Channel_584303BF.TcDUT
{attribute 'GeneratedUsingTerminal: EP2816-0008-0016'}
{attribute addProperty BoxType "EP2816-0008-0016"}
{attribute addProperty Id "Diag_InputAT %I*ARRAY[0..7] OF BOOL8"}
{attribute addProperty CRC "568896300"}
{attribute addProperty Size "8"}
TYPE DO_Inputs_Channel_584303BF EXTENDS InputBase_8311D824 :
STRUCT
	{attribute addProperty Name "Diag_Input"}
	Diag_Input AT %I* : ARRAY[0..7] OF BOOL;
END_STRUCT
END_TYPE

// ---- DUTs/IO/PDOs/DO_Inputs_Device_4E5AF17E.TcDUT
{attribute 'GeneratedUsingTerminal: EP2816-0008-0016'}
{attribute addProperty BoxType "EP2816-0008-0016"}
{attribute addProperty Id "Safe_state_activeAT %I*BOOL1Error_channelAT %I*ARRAY[0..1] OF BOOL2Sync_ErrorAT %I*BOOL1TxPDO_ToggleAT %I*BOOL1"}
{attribute addProperty CRC "3040730866"}
{attribute addProperty Size "5"}
TYPE DO_Inputs_Device_4E5AF17E EXTENDS InputBase_8311D824 :
STRUCT
	{attribute addProperty Name "Safe_state_active"}
	Safe_state_active AT %I* : BOOL;
	{attribute addProperty Name "Error_channel"}
	Error_channel AT %I* : ARRAY[0..1] OF BOOL;
	{attribute addProperty Name "Sync_Error"}
	Sync_Error AT %I* : BOOL;
	{attribute addProperty Name "TxPDO_Toggle"}
	TxPDO_Toggle AT %I* : BOOL;
END_STRUCT
END_TYPE

// ---- DUTs/IO/PDOs/DIG_Outputs_Channel_28AC1A9E.TcDUT
{attribute 'GeneratedUsingTerminal: EP2816-0008-0018'}
{attribute addProperty BoxType "EP2816-0008-0018"}
{attribute addProperty Id "OutputAT %Q*ARRAY[0..7] OF BOOL8"}
{attribute addProperty CRC "1253840710"}
{attribute addProperty Size "8"}
TYPE DIG_Outputs_Channel_28AC1A9E EXTENDS OutputBase_10CEE7DE :
STRUCT
	{attribute addProperty Name "Output"}
	Output AT %Q* : ARRAY[0..7] OF BOOL;
END_STRUCT
END_TYPE

// ---- DUTs/IO/PDOs/DIG_Inputs_Device_27CCC866.TcDUT
{attribute 'GeneratedUsingTerminal: EP2817-0008-0016'}
{attribute addProperty BoxType "EP2817-0008-0016"}
{attribute addProperty Id "Safe_state_activeAT %I*BOOL1Error_channelAT %I*ARRAY[0..2] OF BOOL3Us_UndervoltageAT %I*BOOL1Up_UndervoltageAT %I*BOOL1Sync_errorAT %I*BOOL1TxPDO_ToggleAT %I*BOOL1"}
{attribute addProperty CRC "3987783551"}
{attribute addProperty Size "8"}
TYPE DIG_Inputs_Device_27CCC866 EXTENDS InputBase_8311D824 :
STRUCT
	{attribute addProperty Name "Safe_state_active"}
	Safe_state_active AT %I* : BOOL;
	{attribute addProperty Name "Error_channel"}
	Error_channel AT %I* : ARRAY[0..2] OF BOOL;
	{attribute addProperty Name "Us_Undervoltage"}
	Us_Undervoltage AT %I* : BOOL;
	{attribute addProperty Name "Up_Undervoltage"}
	Up_Undervoltage AT %I* : BOOL;
	{attribute addProperty Name "Sync_error"}
	Sync_error AT %I* : BOOL;
	{attribute addProperty Name "TxPDO_Toggle"}
	TxPDO_Toggle AT %I* : BOOL;
END_STRUCT
END_TYPE

// ---- DUTs/IO/PDOs/AI_Standard_Channel_A8DF64E3.TcDUT
{attribute 'GeneratedUsingTerminal: EP3162-0002-0016'}
{attribute addProperty BoxType "EP3162-0002-0016"}
{attribute addProperty Id "StatusAT %I*Status_B07533568ValueAT %I*INT2"}
{attribute addProperty CRC "2833212643"}
{attribute addProperty Size "10"}
TYPE AI_Standard_Channel_A8DF64E3 EXTENDS InputBase_8311D824 :
STRUCT
	{attribute addProperty Name "Status"}
	Status AT %I* : Status_B0753356;
	{attribute addProperty Name "Value"}
	Value AT %I* : INT;
END_STRUCT
END_TYPE

// ---- DUTs/IO/PDOs/DO_Outputs_C0F4C383.TcDUT
{attribute 'GeneratedUsingTerminal: EP3162-1002-0017'}
{attribute addProperty BoxType "EP3162-1002-0017"}
{attribute addProperty Id "Digital_outputAT %Q*ARRAY[0..1] OF BOOL2"}
{attribute addProperty CRC "2912513055"}
{attribute addProperty Size "2"}
TYPE DO_Outputs_C0F4C383 EXTENDS OutputBase_10CEE7DE :
STRUCT
	{attribute addProperty Name "Digital_output"}
	Digital_output AT %Q* : ARRAY[0..1] OF BOOL;
END_STRUCT
END_TYPE

// ---- DUTs/IO/PDOs/AI_Standard_Channel_4A394481.TcDUT
{attribute 'GeneratedUsingTerminal: EP3174-0002-0016'}
{attribute addProperty BoxType "EP3174-0002-0016"}
{attribute addProperty Id "StatusAT %I*Status_F2CE6D917ValueAT %I*INT2"}
{attribute addProperty CRC "1245267073"}
{attribute addProperty Size "9"}
TYPE AI_Standard_Channel_4A394481 EXTENDS InputBase_8311D824 :
STRUCT
	{attribute addProperty Name "Status"}
	Status AT %I* : Status_F2CE6D91;
	{attribute addProperty Name "Value"}
	Value AT %I* : INT;
END_STRUCT
END_TYPE

// ---- DUTs/IO/PDOs/RTD_RTDInputs_Channel_A8DF64E3.TcDUT
{attribute 'GeneratedUsingTerminal: EP3204-0002-0017'}
{attribute addProperty BoxType "EP3204-0002-0017"}
{attribute addProperty Id "StatusAT %I*Status_B07533568ValueAT %I*INT2"}
{attribute addProperty CRC "2833212643"}
{attribute addProperty Size "10"}
TYPE RTD_RTDInputs_Channel_A8DF64E3 EXTENDS InputBase_8311D824 :
STRUCT
	{attribute addProperty Name "Status"}
	Status AT %I* : Status_B0753356;
	{attribute addProperty Name "Value"}
	Value AT %I* : INT;
END_STRUCT
END_TYPE

// ---- DUTs/IO/PDOs/TC_TCInputs_Channel_A8DF64E3.TcDUT
{attribute 'GeneratedUsingTerminal: EP3314-0002-0016'}
{attribute addProperty BoxType "EP3314-0002-0016"}
{attribute addProperty Id "StatusAT %I*Status_B07533568ValueAT %I*INT2"}
{attribute addProperty CRC "2833212643"}
{attribute addProperty Size "10"}
TYPE TC_TCInputs_Channel_A8DF64E3 EXTENDS InputBase_8311D824 :
STRUCT
	{attribute addProperty Name "Status"}
	Status AT %I* : Status_B0753356;
	{attribute addProperty Name "Value"}
	Value AT %I* : INT;
END_STRUCT
END_TYPE

// ---- DUTs/IO/PDOs/AIBridge_Inputs_555AA1E8.TcDUT
{attribute 'GeneratedUsingTerminal: EP3351-2022-0016'}
{attribute addProperty BoxType "EP3351-2022-0016"}
{attribute addProperty Id "UnderrangeAT %I*BOOL1OverrangeAT %I*BOOL1ErrorAT %I*BOOL1TxPDO_StateAT %I*BOOL1TxPDO_ToggleAT %I*BOOL1ValueAT %I*DINT4"}
{attribute addProperty CRC "1432003048"}
{attribute addProperty Size "9"}
TYPE AIBridge_Inputs_555AA1E8 EXTENDS InputBase_8311D824 :
STRUCT
	{attribute addProperty Name "Underrange"}
	Underrange AT %I* : BOOL;
	{attribute addProperty Name "Overrange"}
	Overrange AT %I* : BOOL;
	{attribute addProperty Name "Error"}
	Error AT %I* : BOOL;
	{attribute addProperty Name "TxPDO_State"}
	TxPDO_State AT %I* : BOOL;
	{attribute addProperty Name "TxPDO_Toggle"}
	TxPDO_Toggle AT %I* : BOOL;
	{attribute addProperty Name "Value"}
	Value AT %I* : DINT;
END_STRUCT
END_TYPE

// ---- DUTs/IO/PDOs/AISupply_Inputs_555AA1E8.TcDUT
{attribute 'GeneratedUsingTerminal: EP3351-2022-0016'}
{attribute addProperty BoxType "EP3351-2022-0016"}
{attribute addProperty Id "UnderrangeAT %I*BOOL1OverrangeAT %I*BOOL1ErrorAT %I*BOOL1TxPDO_StateAT %I*BOOL1TxPDO_ToggleAT %I*BOOL1ValueAT %I*DINT4"}
{attribute addProperty CRC "1432003048"}
{attribute addProperty Size "9"}
TYPE AISupply_Inputs_555AA1E8 EXTENDS InputBase_8311D824 :
STRUCT
	{attribute addProperty Name "Underrange"}
	Underrange AT %I* : BOOL;
	{attribute addProperty Name "Overrange"}
	Overrange AT %I* : BOOL;
	{attribute addProperty Name "Error"}
	Error AT %I* : BOOL;
	{attribute addProperty Name "TxPDO_State"}
	TxPDO_State AT %I* : BOOL;
	{attribute addProperty Name "TxPDO_Toggle"}
	TxPDO_Toggle AT %I* : BOOL;
	{attribute addProperty Name "Value"}
	Value AT %I* : DINT;
END_STRUCT
END_TYPE

// ---- DUTs/IO/PDOs/RMB_Status_C0E100AA.TcDUT
{attribute 'GeneratedUsingTerminal: EP3356-0022-0016'}
{attribute addProperty BoxType "EP3356-0022-0016"}
{attribute addProperty Id "StatusAT %I*Status_7BCDA9217"}
{attribute addProperty CRC "3235971242"}
{attribute addProperty Size "7"}
TYPE RMB_Status_C0E100AA EXTENDS InputBase_8311D824 :
STRUCT
	{attribute addProperty Name "Status"}
	Status AT %I* : Status_7BCDA921;
END_STRUCT
END_TYPE

// ---- DUTs/IO/PDOs/RMB_Value_INT_E9189C4B.TcDUT
{attribute 'GeneratedUsingTerminal: EP3356-0022-0016'}
{attribute addProperty BoxType "EP3356-0022-0016"}
{attribute addProperty Id "ValueAT %I*DINT4"}
{attribute addProperty CRC "3910704203"}
{attribute addProperty Size "4"}
TYPE RMB_Value_INT_E9189C4B EXTENDS InputBase_8311D824 :
STRUCT
	{attribute addProperty Name "Value"}
	Value AT %I* : DINT;
END_STRUCT
END_TYPE

// ---- DUTs/IO/PDOs/RMB_Control_CC49845C.TcDUT
{attribute 'GeneratedUsingTerminal: EP3356-0022-0016'}
{attribute addProperty BoxType "EP3356-0022-0016"}
{attribute addProperty Id "CtrlAT %Q*Ctrl_B9DDD3FF5"}
{attribute addProperty CRC "3427370076"}
{attribute addProperty Size "5"}
TYPE RMB_Control_CC49845C EXTENDS OutputBase_10CEE7DE :
STRUCT
	{attribute addProperty Name "Ctrl"}
	Ctrl AT %Q* : Ctrl_B9DDD3FF;
END_STRUCT
END_TYPE

// ---- DUTs/IO/PDOs/Ch1_Status_75824485.TcDUT
{attribute 'GeneratedUsingTerminal: EP3632-0001-0016'}
{attribute addProperty BoxType "EP3632-0001-0016"}
{attribute addProperty Id "STATUSAT %I*STATUS_B07533568"}
{attribute addProperty CRC "1971471493"}
{attribute addProperty Size "8"}
TYPE Ch1_Status_75824485 EXTENDS InputBase_8311D824 :
STRUCT
	{attribute addProperty Name "STATUS"}
	STATUS AT %I* : STATUS_B0753356;
END_STRUCT
END_TYPE

// ---- DUTs/IO/PDOs/Ch1_Sample_A71DD501.TcDUT
{attribute 'GeneratedUsingTerminal: EP3632-0001-0016'}
{attribute addProperty BoxType "EP3632-0001-0016"}
{attribute addProperty Id "Ch1_ValueAT %I*INT2"}
{attribute addProperty CRC "2803750145"}
{attribute addProperty Size "2"}
TYPE Ch1_Sample_A71DD501 EXTENDS InputBase_8311D824 :
STRUCT
	{attribute addProperty Name "Ch1_Value"}
	Ch1_Value AT %I* : INT;
END_STRUCT
END_TYPE

// ---- DUTs/IO/PDOs/Ch2_Status_75824485.TcDUT
{attribute 'GeneratedUsingTerminal: EP3632-0001-0016'}
{attribute addProperty BoxType "EP3632-0001-0016"}
{attribute addProperty Id "STATUSAT %I*STATUS_B07533568"}
{attribute addProperty CRC "1971471493"}
{attribute addProperty Size "8"}
TYPE Ch2_Status_75824485 EXTENDS InputBase_8311D824 :
STRUCT
	{attribute addProperty Name "STATUS"}
	STATUS AT %I* : STATUS_B0753356;
END_STRUCT
END_TYPE

// ---- DUTs/IO/PDOs/Ch2_Sample_9F6886E6.TcDUT
{attribute 'GeneratedUsingTerminal: EP3632-0001-0016'}
{attribute addProperty BoxType "EP3632-0001-0016"}
{attribute addProperty Id "Ch2_ValueAT %I*INT2"}
{attribute addProperty CRC "2674427622"}
{attribute addProperty Size "2"}
TYPE Ch2_Sample_9F6886E6 EXTENDS InputBase_8311D824 :
STRUCT
	{attribute addProperty Name "Ch2_Value"}
	Ch2_Value AT %I* : INT;
END_STRUCT
END_TYPE

// ---- DUTs/IO/PDOs/NextSync1Time_9AFDC275.TcDUT
{attribute 'GeneratedUsingTerminal: EP3632-0001-0016'}
{attribute addProperty BoxType "EP3632-0001-0016"}
{attribute addProperty Id "StartTimeNextLatchAT %I*ULINT8"}
{attribute addProperty CRC "2600321653"}
{attribute addProperty Size "8"}
TYPE NextSync1Time_9AFDC275 EXTENDS InputBase_8311D824 :
STRUCT
	{attribute addProperty Name "StartTimeNextLatch"}
	StartTimeNextLatch AT %I* : ULINT;
END_STRUCT
END_TYPE

// ---- DUTs/IO/PDOs/Sample_Count_EA88CAD9.TcDUT
{attribute 'GeneratedUsingTerminal: EP3632-0001-0016'}
{attribute addProperty BoxType "EP3632-0001-0016"}
{attribute addProperty Id "Sample_CountAT %I*UINT2"}
{attribute addProperty CRC "3934833369"}
{attribute addProperty Size "2"}
TYPE Sample_Count_EA88CAD9 EXTENDS InputBase_8311D824 :
STRUCT
	{attribute addProperty Name "Sample_Count"}
	Sample_Count AT %I* : UINT;
END_STRUCT
END_TYPE

// ---- DUTs/IO/PDOs/InfoData_BEF6B88E.TcDUT
{attribute 'GeneratedUsingTerminal: EP3632-0001-0016'}
{attribute addProperty BoxType "EP3632-0001-0016"}
{attribute addProperty Id "AdsAddrAT %I*AMSADDR8DcOutputShiftAT %I*DINT4DcInputShiftAT %I*DINT4StateAT %I*UINT2"}
{attribute addProperty CRC "3203840142"}
{attribute addProperty Size "18"}
TYPE InfoData_BEF6B88E EXTENDS InputBase_8311D824 :
STRUCT
	{attribute addProperty Name "AdsAddr"}
	AdsAddr AT %I* : AMSADDR;
	{attribute addProperty Name "DcOutputShift"}
	DcOutputShift AT %I* : DINT;
	{attribute addProperty Name "DcInputShift"}
	DcInputShift AT %I* : DINT;
	{attribute addProperty Name "State"}
	State AT %I* : UINT;
END_STRUCT
END_TYPE

// ---- DUTs/IO/PDOs/DIG_Inputs_697E0EF2.TcDUT
{attribute 'GeneratedUsingTerminal: EP3744-0041-0016'}
{attribute addProperty BoxType "EP3744-0041-0016"}
{attribute addProperty Id "InputAT %I*ARRAY[0..5] OF BOOL6"}
{attribute addProperty CRC "390650255"}
{attribute addProperty Size "6"}
TYPE DIG_Inputs_697E0EF2 EXTENDS InputBase_8311D824 :
STRUCT
	{attribute addProperty Name "Input"}
	Input AT %I* : ARRAY[0..5] OF BOOL;
END_STRUCT
END_TYPE

// ---- DUTs/IO/PDOs/AI_Inputs_Channel_45213104.TcDUT
{attribute 'GeneratedUsingTerminal: EP3744-0041-0016'}
{attribute addProperty BoxType "EP3744-0041-0016"}
{attribute addProperty Id "StatusAT %I*Status_F2CE6D917ValueAT %I*DINT4"}
{attribute addProperty CRC "1159803140"}
{attribute addProperty Size "11"}
TYPE AI_Inputs_Channel_45213104 EXTENDS InputBase_8311D824 :
STRUCT
	{attribute addProperty Name "Status"}
	Status AT %I* : Status_F2CE6D91;
	{attribute addProperty Name "Value"}
	Value AT %I* : DINT;
END_STRUCT
END_TYPE

// ---- DUTs/IO/PDOs/DEV_Inputs_Device_5F4E175E.TcDUT
{attribute 'GeneratedUsingTerminal: EP3744-0041-0016'}
{attribute addProperty BoxType "EP3744-0041-0016"}
{attribute addProperty Id "Safe_State_ActiveAT %I*BOOL1Sync_errorAT %I*BOOL1Undervoltage_UsAT %I*BOOL1Undervoltage_UpAT %I*BOOL1TxPDO_ToggleAT %I*BOOL1"}
{attribute addProperty CRC "1598953310"}
{attribute addProperty Size "5"}
TYPE DEV_Inputs_Device_5F4E175E EXTENDS InputBase_8311D824 :
STRUCT
	{attribute addProperty Name "Safe_State_Active"}
	Safe_State_Active AT %I* : BOOL;
	{attribute addProperty Name "Sync_error"}
	Sync_error AT %I* : BOOL;
	{attribute addProperty Name "Undervoltage_Us"}
	Undervoltage_Us AT %I* : BOOL;
	{attribute addProperty Name "Undervoltage_Up"}
	Undervoltage_Up AT %I* : BOOL;
	{attribute addProperty Name "TxPDO_Toggle"}
	TxPDO_Toggle AT %I* : BOOL;
END_STRUCT
END_TYPE

// ---- DUTs/IO/PDOs/DIG_Outputs_DE230DD5.TcDUT
{attribute 'GeneratedUsingTerminal: EP3744-0041-0016'}
{attribute addProperty BoxType "EP3744-0041-0016"}
{attribute addProperty Id "OutputAT %Q*ARRAY[0..1] OF BOOL2"}
{attribute addProperty CRC "2036329114"}
{attribute addProperty Size "2"}
TYPE DIG_Outputs_DE230DD5 EXTENDS OutputBase_10CEE7DE :
STRUCT
	{attribute addProperty Name "Output"}
	Output AT %Q* : ARRAY[0..1] OF BOOL;
END_STRUCT
END_TYPE

// ---- DUTs/IO/PDOs/DEV_Outputs_Device_59FFD247.TcDUT
{attribute 'GeneratedUsingTerminal: EP3744-0041-0016'}
{attribute addProperty BoxType "EP3744-0041-0016"}
{attribute addProperty Id "Set_safe_stateAT %Q*BOOL1"}
{attribute addProperty CRC "1509937735"}
{attribute addProperty Size "1"}
TYPE DEV_Outputs_Device_59FFD247 EXTENDS OutputBase_10CEE7DE :
STRUCT
	{attribute addProperty Name "Set_safe_state"}
	Set_safe_state AT %Q* : BOOL;
END_STRUCT
END_TYPE

// ---- DUTs/IO/PDOs/AI_Inputs_Channel_5A86716D.TcDUT
{attribute 'GeneratedUsingTerminal: EP3752-0000-0017'}
{attribute addProperty BoxType "EP3752-0000-0017"}
{attribute addProperty Id "StatusAT %I*Status_8F1D55D83ValueAT %I*INT2"}
{attribute addProperty CRC "1518760301"}
{attribute addProperty Size "5"}
TYPE AI_Inputs_Channel_5A86716D EXTENDS InputBase_8311D824 :
STRUCT
	{attribute addProperty Name "Status"}
	Status AT %I* : Status_8F1D55D8;
	{attribute addProperty Name "Value"}
	Value AT %I* : INT;
END_STRUCT
END_TYPE

// ---- DUTs/IO/PDOs/AO_Output_Channel_BA7EBB7C.TcDUT
{attribute 'GeneratedUsingTerminal: EP4174-0002-0016'}
{attribute addProperty BoxType "EP4174-0002-0016"}
{attribute addProperty Id "Analog_outputAT %Q*INT2"}
{attribute addProperty CRC "3128867708"}
{attribute addProperty Size "2"}
TYPE AO_Output_Channel_BA7EBB7C EXTENDS OutputBase_10CEE7DE :
STRUCT
	{attribute addProperty Name "Analog_output"}
	Analog_output AT %Q* : INT;
END_STRUCT
END_TYPE

// ---- DUTs/IO/PDOs/DI_Inputs_1F3A9325.TcDUT
{attribute 'GeneratedUsingTerminal: EP4314-1002-0016'}
{attribute addProperty BoxType "EP4314-1002-0016"}
{attribute addProperty Id "InputAT %I*ARRAY[0..1] OF BOOL2TxPDO_StateAT %I*BOOL1TxPDO_ToggleAT %I*BOOL1"}
{attribute addProperty CRC "2573189997"}
{attribute addProperty Size "4"}
TYPE DI_Inputs_1F3A9325 EXTENDS InputBase_8311D824 :
STRUCT
	{attribute addProperty Name "Input"}
	Input AT %I* : ARRAY[0..1] OF BOOL;
	{attribute addProperty Name "TxPDO_State"}
	TxPDO_State AT %I* : BOOL;
	{attribute addProperty Name "TxPDO_Toggle"}
	TxPDO_Toggle AT %I* : BOOL;
END_STRUCT
END_TYPE

// ---- DUTs/IO/PDOs/AI_TxPDO_Map_Standard_Channel_A8DF64E3.TcDUT
{attribute 'GeneratedUsingTerminal: EP4374-0002-0016'}
{attribute addProperty BoxType "EP4374-0002-0016"}
{attribute addProperty Id "StatusAT %I*Status_B07533568ValueAT %I*INT2"}
{attribute addProperty CRC "2833212643"}
{attribute addProperty Size "10"}
TYPE AI_TxPDO_Map_Standard_Channel_A8DF64E3 EXTENDS InputBase_8311D824 :
STRUCT
	{attribute addProperty Name "Status"}
	Status AT %I* : Status_B0753356;
	{attribute addProperty Name "Value"}
	Value AT %I* : INT;
END_STRUCT
END_TYPE

// ---- DUTs/IO/PDOs/AI_Inputs_Channel_A8DF64E3.TcDUT
{attribute 'GeneratedUsingTerminal: EP4374-0002-0017'}
{attribute addProperty BoxType "EP4374-0002-0017"}
{attribute addProperty Id "StatusAT %I*Status_B07533568ValueAT %I*INT2"}
{attribute addProperty CRC "2833212643"}
{attribute addProperty Size "10"}
TYPE AI_Inputs_Channel_A8DF64E3 EXTENDS InputBase_8311D824 :
STRUCT
	{attribute addProperty Name "Status"}
	Status AT %I* : Status_B0753356;
	{attribute addProperty Name "Value"}
	Value AT %I* : INT;
END_STRUCT
END_TYPE

// ---- DUTs/IO/PDOs/DI_X03_Pin4_Input_830843C1.TcDUT
{attribute 'GeneratedUsingTerminal: EP4378-1022-0017'}
{attribute addProperty BoxType "EP4378-1022-0017"}
{attribute addProperty Id "InputAT %I*BOOL1"}
{attribute addProperty CRC "2198356929"}
{attribute addProperty Size "1"}
TYPE DI_X03_Pin4_Input_830843C1 EXTENDS InputBase_8311D824 :
STRUCT
	{attribute addProperty Name "Input"}
	Input AT %I* : BOOL;
END_STRUCT
END_TYPE

// ---- DUTs/IO/PDOs/DI_X04_Pin4_Input_830843C1.TcDUT
{attribute 'GeneratedUsingTerminal: EP4378-1022-0017'}
{attribute addProperty BoxType "EP4378-1022-0017"}
{attribute addProperty Id "InputAT %I*BOOL1"}
{attribute addProperty CRC "2198356929"}
{attribute addProperty Size "1"}
TYPE DI_X04_Pin4_Input_830843C1 EXTENDS InputBase_8311D824 :
STRUCT
	{attribute addProperty Name "Input"}
	Input AT %I* : BOOL;
END_STRUCT
END_TYPE

// ---- DUTs/IO/PDOs/DI_X05_Pin4_Input_830843C1.TcDUT
{attribute 'GeneratedUsingTerminal: EP4378-1022-0017'}
{attribute addProperty BoxType "EP4378-1022-0017"}
{attribute addProperty Id "InputAT %I*BOOL1"}
{attribute addProperty CRC "2198356929"}
{attribute addProperty Size "1"}
TYPE DI_X05_Pin4_Input_830843C1 EXTENDS InputBase_8311D824 :
STRUCT
	{attribute addProperty Name "Input"}
	Input AT %I* : BOOL;
END_STRUCT
END_TYPE

// ---- DUTs/IO/PDOs/DI_X06_Pin4_Input_830843C1.TcDUT
{attribute 'GeneratedUsingTerminal: EP4378-1022-0017'}
{attribute addProperty BoxType "EP4378-1022-0017"}
{attribute addProperty Id "InputAT %I*BOOL1"}
{attribute addProperty CRC "2198356929"}
{attribute addProperty Size "1"}
TYPE DI_X06_Pin4_Input_830843C1 EXTENDS InputBase_8311D824 :
STRUCT
	{attribute addProperty Name "Input"}
	Input AT %I* : BOOL;
END_STRUCT
END_TYPE

// ---- DUTs/IO/PDOs/DI_X07_Pin4_Input_830843C1.TcDUT
{attribute 'GeneratedUsingTerminal: EP4378-1022-0017'}
{attribute addProperty BoxType "EP4378-1022-0017"}
{attribute addProperty Id "InputAT %I*BOOL1"}
{attribute addProperty CRC "2198356929"}
{attribute addProperty Size "1"}
TYPE DI_X07_Pin4_Input_830843C1 EXTENDS InputBase_8311D824 :
STRUCT
	{attribute addProperty Name "Input"}
	Input AT %I* : BOOL;
END_STRUCT
END_TYPE

// ---- DUTs/IO/PDOs/DI_X08_Pin4_Input_830843C1.TcDUT
{attribute 'GeneratedUsingTerminal: EP4378-1022-0017'}
{attribute addProperty BoxType "EP4378-1022-0017"}
{attribute addProperty Id "InputAT %I*BOOL1"}
{attribute addProperty CRC "2198356929"}
{attribute addProperty Size "1"}
TYPE DI_X08_Pin4_Input_830843C1 EXTENDS InputBase_8311D824 :
STRUCT
	{attribute addProperty Name "Input"}
	Input AT %I* : BOOL;
END_STRUCT
END_TYPE

// ---- DUTs/IO/PDOs/AI_X01_Pin2_Standard_A8DF64E3.TcDUT
{attribute 'GeneratedUsingTerminal: EP4378-1022-0017'}
{attribute addProperty BoxType "EP4378-1022-0017"}
{attribute addProperty Id "StatusAT %I*Status_B07533568ValueAT %I*INT2"}
{attribute addProperty CRC "2833212643"}
{attribute addProperty Size "10"}
TYPE AI_X01_Pin2_Standard_A8DF64E3 EXTENDS InputBase_8311D824 :
STRUCT
	{attribute addProperty Name "Status"}
	Status AT %I* : Status_B0753356;
	{attribute addProperty Name "Value"}
	Value AT %I* : INT;
END_STRUCT
END_TYPE

// ---- DUTs/IO/PDOs/AI_X02_Pin2_Standard_A8DF64E3.TcDUT
{attribute 'GeneratedUsingTerminal: EP4378-1022-0017'}
{attribute addProperty BoxType "EP4378-1022-0017"}
{attribute addProperty Id "StatusAT %I*Status_B07533568ValueAT %I*INT2"}
{attribute addProperty CRC "2833212643"}
{attribute addProperty Size "10"}
TYPE AI_X02_Pin2_Standard_A8DF64E3 EXTENDS InputBase_8311D824 :
STRUCT
	{attribute addProperty Name "Status"}
	Status AT %I* : Status_B0753356;
	{attribute addProperty Name "Value"}
	Value AT %I* : INT;
END_STRUCT
END_TYPE

// ---- DUTs/IO/PDOs/AI_X05_Pin2_Standard_A8DF64E3.TcDUT
{attribute 'GeneratedUsingTerminal: EP4378-1022-0017'}
{attribute addProperty BoxType "EP4378-1022-0017"}
{attribute addProperty Id "StatusAT %I*Status_B07533568ValueAT %I*INT2"}
{attribute addProperty CRC "2833212643"}
{attribute addProperty Size "10"}
TYPE AI_X05_Pin2_Standard_A8DF64E3 EXTENDS InputBase_8311D824 :
STRUCT
	{attribute addProperty Name "Status"}
	Status AT %I* : Status_B0753356;
	{attribute addProperty Name "Value"}
	Value AT %I* : INT;
END_STRUCT
END_TYPE

// ---- DUTs/IO/PDOs/AI_X06_Pin2_Standard_A8DF64E3.TcDUT
{attribute 'GeneratedUsingTerminal: EP4378-1022-0017'}
{attribute addProperty BoxType "EP4378-1022-0017"}
{attribute addProperty Id "StatusAT %I*Status_B07533568ValueAT %I*INT2"}
{attribute addProperty CRC "2833212643"}
{attribute addProperty Size "10"}
TYPE AI_X06_Pin2_Standard_A8DF64E3 EXTENDS InputBase_8311D824 :
STRUCT
	{attribute addProperty Name "Status"}
	Status AT %I* : Status_B0753356;
	{attribute addProperty Name "Value"}
	Value AT %I* : INT;
END_STRUCT
END_TYPE

// ---- DUTs/IO/PDOs/DO_X01_Pin4_Output_42CA91F7.TcDUT
{attribute 'GeneratedUsingTerminal: EP4378-1022-0017'}
{attribute addProperty BoxType "EP4378-1022-0017"}
{attribute addProperty Id "OutputAT %Q*BOOL1"}
{attribute addProperty CRC "1120571895"}
{attribute addProperty Size "1"}
TYPE DO_X01_Pin4_Output_42CA91F7 EXTENDS OutputBase_10CEE7DE :
STRUCT
	{attribute addProperty Name "Output"}
	Output AT %Q* : BOOL;
END_STRUCT
END_TYPE

// ---- DUTs/IO/PDOs/DO_X02_Pin4_Output_42CA91F7.TcDUT
{attribute 'GeneratedUsingTerminal: EP4378-1022-0017'}
{attribute addProperty BoxType "EP4378-1022-0017"}
{attribute addProperty Id "OutputAT %Q*BOOL1"}
{attribute addProperty CRC "1120571895"}
{attribute addProperty Size "1"}
TYPE DO_X02_Pin4_Output_42CA91F7 EXTENDS OutputBase_10CEE7DE :
STRUCT
	{attribute addProperty Name "Output"}
	Output AT %Q* : BOOL;
END_STRUCT
END_TYPE

// ---- DUTs/IO/PDOs/DO_X05_Pin4_Output_42CA91F7.TcDUT
{attribute 'GeneratedUsingTerminal: EP4378-1022-0017'}
{attribute addProperty BoxType "EP4378-1022-0017"}
{attribute addProperty Id "OutputAT %Q*BOOL1"}
{attribute addProperty CRC "1120571895"}
{attribute addProperty Size "1"}
TYPE DO_X05_Pin4_Output_42CA91F7 EXTENDS OutputBase_10CEE7DE :
STRUCT
	{attribute addProperty Name "Output"}
	Output AT %Q* : BOOL;
END_STRUCT
END_TYPE

